// TwinCAT 3 PLC project PLC
// ProgramVersion: 3.1.4024.0
// libraries:
//   EfficientIO Communicator, * (EfficientIO)
//   EfficientIO Energy Basic, * (EfficientIO)
//   EfficientIO ModbusTCP, * (EfficientIO)
//   Lynus Persistent Data V1, * (Lynus AG)
//   Lynus Standards, * (Lynus AG)
//   Tc2_EtherCAT, * (Beckhoff Automation GmbH)
//   Tc2_ModbusSrv, * (Beckhoff Automation GmbH)
//   Tc2_Standard, * (Beckhoff Automation GmbH)
//   Tc2_System, * (Beckhoff Automation GmbH)
//   Tc2_Utilities, * (Beckhoff Automation GmbH)
//   Tc3_Module, * (Beckhoff Automation GmbH)
// project tree:
//   / FastTask.TcTTO, MiddleTask.TcTTO, SlowTask.TcTTO
//   FBs/EL3443_DPM/DUTs/ E_EL3443_DPM_Phase.TcDUT (not stored), E_EL3443_DPM_Total.TcDUT (not stored), MDP5001_341_7CD731EE.TcDUT (not stored), MDP5001_341_I_7CD731EE.TcDUT (not stored), MDP5001_341_O_7CD731EE.TcDUT (not stored), ST_EL3443_DPM_MUX_REAL.TcDUT (not stored), ST_EL3443_DPM_MUX_ULINT.TcDUT (not stored), ST_EL3443_DPM_StatusLx.TcDUT (not stored), ST_EL3443_DPM_StatusTotal.TcDUT (not stored), ST_EL3443_DPM_VariantLx.TcDUT, ST_EL3443_DPM_VariantTotal.TcDUT (not stored), ST_EL3443_DPM_VariantValues.TcDUT (not stored)
//   FBs/EL3443_DPM/ FB_EL3443_DPM.TcPOU (not stored)
//   FBs/EL3446 FW02 or higher/DUTs/ E_EL3446_Phase.TcDUT (not stored), MDP5001_342_066CA8C6.TcDUT, MDP5001_342_I_066CA8C6.TcDUT (not stored), MDP5001_342_O_066CA8C6.TcDUT (not stored), ST_EL3446_MUX_REAL.TcDUT (not stored), ST_EL3446_MUX_ULINT.TcDUT (not stored), ST_EL3446_StatusIx.TcDUT (not stored), ST_EL3446_VariantIx.TcDUT (not stored), ST_EL3446_VariantValues.TcDUT (not stored)
//   FBs/EL3446 FW02 or higher/ FB_EL3446.TcPOU (not stored)
//   FBs/ FB_CoE_EL3443.TcPOU (not stored), FB_CoE_EL3446.TcPOU, FB_ECS_Keba_P30_noWrite.TcPOU, FB_EM_Beckhoff_EL3443.TcPOU, FB_EM_Beckhoff_EL3446.TcPOU, FB_ModBus_100Registers_FC3_inclID.TcPOU, FB_Symo_PV_Inverter_FLOAT_1_DM_30_Inverter_1.TcPOU, FB_Symo_PV_Inverter_INT_1_DM_30_Inverter_1.TcPOU
//   POUs/ prgComEffIO.TcPOU, prgCS.TcPOU, prgEM.TcPOU, prgHW.TcPOU, prgPersistent.TcPOU, prgPV.TcPOU, prgRWEffIO.TcPOU, prgVarEffIO.TcPOU
// real-time tasks:
//   TASK FastTask: cycle T#5ms, priority 19, ADS port 351
//   TASK MiddleTask: cycle T#10ms, priority 20, ADS port 352
//   TASK SlowTask: cycle T#20ms, priority 21, ADS port 353
// I/O:
//   DEVICE Gerät 1 (EtherCAT), AmsNetId 5.114.133.36.2.1
//     Klemme 1 (EK1200) [EK1200-5000 EtherCAT Netzteil (2A E-Bus)]
//       Klemme 2 (EL3443) [EL3443 3K. Leistungsmessung]
//       Klemme 3 (EL3446) [EL3446 DPM 6 K. Strommessklemme]
//       Klemme 4 (EL3446) [EL3446 DPM 6 K. Strommessklemme]
//       Klemme 5 (EL3446) [EL3446 DPM 6 K. Strommessklemme]
//       Klemme 6 (EL3446) [EL3446 DPM 6 K. Strommessklemme]
//       Klemme 7 (EL9011) [EL9011 Endklemme]
// variable links:
//   PLC/PLC Instance <-> Device 1 (EtherCAT)/Term 1 (EK1200)/Term 2 (EL3443)
//     FastTask Inputs/prgHW.MDP5001_341_DPM_Data_Data_{1..20} <-> DPM Data/Data {1..20}  (20 links)
//     FastTask Inputs/prgHW.MDP5001_341_L1_Basic_Current <-> L1 Basic/Current
//     FastTask Inputs/prgHW.MDP5001_341_L2_Basic_Current <-> L2 Basic/Current
//     FastTask Inputs/prgHW.MDP5001_341_L3_Basic_Current <-> L3 Basic/Current
//     FastTask Inputs/prgHW.MDP5001_341_L1_Basic_Voltage <-> L1 Basic/Voltage
//     FastTask Inputs/prgHW.MDP5001_341_L2_Basic_Voltage <-> L2 Basic/Voltage
//     FastTask Inputs/prgHW.MDP5001_341_L3_Basic_Voltage <-> L3 Basic/Voltage
//     FastTask Inputs/prgHW.MDP5001_341_L1_Power_Active_Power <-> L1 Power/Active Power
//     FastTask Inputs/prgHW.MDP5001_341_L2_Power_Active_Power <-> L2 Power/Active Power
//     FastTask Inputs/prgHW.MDP5001_341_L3_Power_Active_Power <-> L3 Power/Active Power
//     FastTask Inputs/prgHW.MDP5001_341_L1_Power_Apparent_Power <-> L1 Power/Apparent Power
//     FastTask Inputs/prgHW.MDP5001_341_L2_Power_Apparent_Power <-> L2 Power/Apparent Power
//     FastTask Inputs/prgHW.MDP5001_341_L3_Power_Apparent_Power <-> L3 Power/Apparent Power
//     FastTask Inputs/prgHW.MDP5001_341_L1_Power_Power_Factor <-> L1 Power/Power Factor
//     FastTask Inputs/prgHW.MDP5001_341_L2_Power_Power_Factor <-> L2 Power/Power Factor
//     FastTask Inputs/prgHW.MDP5001_341_L3_Power_Power_Factor <-> L3 Power/Power Factor
//     FastTask Inputs/prgHW.MDP5001_341_L1_Power_Reactive_Power <-> L1 Power/Reactive Power
//     FastTask Inputs/prgHW.MDP5001_341_L2_Power_Reactive_Power <-> L2 Power/Reactive Power
//     FastTask Inputs/prgHW.MDP5001_341_L3_Power_Reactive_Power <-> L3 Power/Reactive Power
//     FastTask Inputs/prgHW.MDP5001_341_L1_Status_Current_Guard_Error <-> L1 Status/Current Guard Error
//     FastTask Inputs/prgHW.MDP5001_341_L2_Status_Current_Guard_Error <-> L2 Status/Current Guard Error
//     FastTask Inputs/prgHW.MDP5001_341_L3_Status_Current_Guard_Error <-> L3 Status/Current Guard Error
//     FastTask Inputs/prgHW.MDP5001_341_L1_Status_Current_Guard_Warning <-> L1 Status/Current Guard Warning
//     FastTask Inputs/prgHW.MDP5001_341_L2_Status_Current_Guard_Warning <-> L2 Status/Current Guard Warning
//     FastTask Inputs/prgHW.MDP5001_341_L3_Status_Current_Guard_Warning <-> L3 Status/Current Guard Warning
//     FastTask Inputs/prgHW.MDP5001_341_L1_Status_Inaccurate_Current <-> L1 Status/Inaccurate Current
//     FastTask Inputs/prgHW.MDP5001_341_L2_Status_Inaccurate_Current <-> L2 Status/Inaccurate Current
//     FastTask Inputs/prgHW.MDP5001_341_L3_Status_Inaccurate_Current <-> L3 Status/Inaccurate Current
//     FastTask Inputs/prgHW.MDP5001_341_L1_Status_Inaccurate_Voltage <-> L1 Status/Inaccurate Voltage
//     FastTask Inputs/prgHW.MDP5001_341_L2_Status_Inaccurate_Voltage <-> L2 Status/Inaccurate Voltage
//     FastTask Inputs/prgHW.MDP5001_341_L3_Status_Inaccurate_Voltage <-> L3 Status/Inaccurate Voltage
//     FastTask Inputs/prgHW.MDP5001_341_L1_Status_Overcurrent <-> L1 Status/Overcurrent
//     FastTask Inputs/prgHW.MDP5001_341_L2_Status_Overcurrent <-> L2 Status/Overcurrent
//     FastTask Inputs/prgHW.MDP5001_341_L3_Status_Overcurrent <-> L3 Status/Overcurrent
//     FastTask Inputs/prgHW.MDP5001_341_L1_Status_Overvoltage <-> L1 Status/Overvoltage
//     FastTask Inputs/prgHW.MDP5001_341_L2_Status_Overvoltage <-> L2 Status/Overvoltage
//     FastTask Inputs/prgHW.MDP5001_341_L3_Status_Overvoltage <-> L3 Status/Overvoltage
//     FastTask Inputs/prgHW.MDP5001_341_L1_Status_TxPDO_Toggle <-> L1 Status/TxPDO Toggle
//     FastTask Inputs/prgHW.MDP5001_341_L2_Status_TxPDO_Toggle <-> L2 Status/TxPDO Toggle
//     FastTask Inputs/prgHW.MDP5001_341_L3_Status_TxPDO_Toggle <-> L3 Status/TxPDO Toggle
//     FastTask Inputs/prgHW.MDP5001_341_L1_Status_Voltage_Guard_Error <-> L1 Status/Voltage Guard Error
//     FastTask Inputs/prgHW.MDP5001_341_L2_Status_Voltage_Guard_Error <-> L2 Status/Voltage Guard Error
//     FastTask Inputs/prgHW.MDP5001_341_L3_Status_Voltage_Guard_Error <-> L3 Status/Voltage Guard Error
//     FastTask Inputs/prgHW.MDP5001_341_L1_Status_Voltage_Guard_Warning <-> L1 Status/Voltage Guard Warning
//     FastTask Inputs/prgHW.MDP5001_341_L2_Status_Voltage_Guard_Warning <-> L2 Status/Voltage Guard Warning
//     FastTask Inputs/prgHW.MDP5001_341_L3_Status_Voltage_Guard_Warning <-> L3 Status/Voltage Guard Warning
//     FastTask Inputs/prgHW.MDP5001_341_L1_Status_Voltage_Sign_Bit <-> L1 Status/Voltage Sign Bit
//     FastTask Inputs/prgHW.MDP5001_341_L2_Status_Voltage_Sign_Bit <-> L2 Status/Voltage Sign Bit
//     FastTask Inputs/prgHW.MDP5001_341_L3_Status_Voltage_Sign_Bit <-> L3 Status/Voltage Sign Bit
//     FastTask Inputs/prgHW.MDP5001_341_Total_Basic_Calculated_Neutral_Line_Current <-> Total Basic/Calculated Neutral Line Current
//     FastTask Inputs/prgHW.MDP5001_341_Total_Basic_Frequency <-> Total Basic/Frequency
//     FastTask Inputs/prgHW.MDP5001_341_Total_Basic_Power_Factor <-> Total Basic/Power Factor
//     FastTask Inputs/prgHW.MDP5001_341_Total_Status_Active_Power_Guard_Error <-> Total Status/Active Power Guard Error
//     FastTask Inputs/prgHW.MDP5001_341_Total_Status_Active_Power_Guard_Warning <-> Total Status/Active Power Guard Warning
//     FastTask Inputs/prgHW.MDP5001_341_Total_Status_Apparent_Power_Guard_Error <-> Total Status/Apparent Power Guard Error
//     FastTask Inputs/prgHW.MDP5001_341_Total_Status_Apparent_Power_Guard_Warning <-> Total Status/Apparent Power Guard Warning
//     FastTask Inputs/prgHW.MDP5001_341_Total_Status_Frequency_Guard_Error <-> Total Status/Frequency Guard Error
//     FastTask Inputs/prgHW.MDP5001_341_Total_Status_Frequency_Guard_Warning <-> Total Status/Frequency Guard Warning
//     FastTask Inputs/prgHW.MDP5001_341_Total_Status_Grid_Direction <-> Total Status/Grid Direction
//     FastTask Inputs/prgHW.MDP5001_341_Total_Status_Neutral_Current_Guard_Error <-> Total Status/Neutral Current Guard Error
//     FastTask Inputs/prgHW.MDP5001_341_Total_Status_Neutral_Current_Guard_Warning <-> Total Status/Neutral Current Guard Warning
//     FastTask Inputs/prgHW.MDP5001_341_Total_Status_Power_Quality_Factor <-> Total Status/Power Quality Factor
//     FastTask Inputs/prgHW.MDP5001_341_Total_Status_Power_Quality_Guard_Error <-> Total Status/Power Quality Guard Error
//     FastTask Inputs/prgHW.MDP5001_341_Total_Status_Power_Quality_Guard_Warning <-> Total Status/Power Quality Guard Warning
//     FastTask Inputs/prgHW.MDP5001_341_Total_Status_System_State <-> Total Status/System State
//     FastTask Inputs/prgHW.MDP5001_341_Total_Status_TxPDO_State <-> Total Status/TxPDO State
//     FastTask Inputs/prgHW.MDP5001_341_Total_Status_TxPDO_Toggle <-> Total Status/TxPDO Toggle
//     FastTask Inputs/prgHW.MDP5001_341_Total_Variant_Value_In_Index_1_REAL <-> Total Variant Value In/Index 1 REAL
//     FastTask Inputs/prgHW.MDP5001_341_Total_Variant_Value_In_Index_2_REAL <-> Total Variant Value In/Index 2 REAL
//     FastTask Inputs/prgHW.MDP5001_341_Total_Variant_Value_In_Index_3_REAL <-> Total Variant Value In/Index 3 REAL
//     FastTask Inputs/prgHW.MDP5001_341_Total_Variant_Value_In_Index_4_ULINT <-> Total Variant Value In/Index 4 ULINT
//     FastTask Inputs/prgHW.MDP5001_341_Total_Variant_Value_In_TxPDO_Toggle <-> Total Variant Value In/TxPDO Toggle
//     FastTask Inputs/prgHW.MDP5001_341_Total_Variant_Value_In_Value_1_REAL <-> Total Variant Value In/Value 1 REAL
//     FastTask Inputs/prgHW.MDP5001_341_Total_Variant_Value_In_Value_2_REAL <-> Total Variant Value In/Value 2 REAL
//     FastTask Inputs/prgHW.MDP5001_341_Total_Variant_Value_In_Value_3_REAL <-> Total Variant Value In/Value 3 REAL
//     FastTask Inputs/prgHW.MDP5001_341_Total_Variant_Value_In_Value_4_ULINT <-> Total Variant Value In/Value 4 ULINT
//     FastTask Outputs/prgHW.MDP5001_341_Total_Interval_Reset_Interval <-> Total Interval/Reset Interval
//     FastTask Outputs/prgHW.MDP5001_341_Total_Variant_Value_Out_Index_1_REAL <-> Total Variant Value Out/Index 1 REAL
//     FastTask Outputs/prgHW.MDP5001_341_Total_Variant_Value_Out_Index_2_REAL <-> Total Variant Value Out/Index 2 REAL
//     FastTask Outputs/prgHW.MDP5001_341_Total_Variant_Value_Out_Index_3_REAL <-> Total Variant Value Out/Index 3 REAL
//     FastTask Outputs/prgHW.MDP5001_341_Total_Variant_Value_Out_Index_4_ULINT <-> Total Variant Value Out/Index 4 ULINT
//   PLC/PLC Instance <-> Device 1 (EtherCAT)/Term 1 (EK1200)/Term 3 (EL3446)
//     FastTask Inputs/prgHW.MDP5001_342_DPM_Variant_Value_In_Index_1_REAL_1 <-> DPM Variant Value In/Index 1 REAL
//     FastTask Inputs/prgHW.MDP5001_342_DPM_Variant_Value_In_Index_2_REAL_1 <-> DPM Variant Value In/Index 2 REAL
//     FastTask Inputs/prgHW.MDP5001_342_DPM_Variant_Value_In_Index_3_REAL_1 <-> DPM Variant Value In/Index 3 REAL
//     FastTask Inputs/prgHW.MDP5001_342_DPM_Variant_Value_In_Index_4_ULINT_1 <-> DPM Variant Value In/Index 4 ULINT
//     FastTask Inputs/prgHW.MDP5001_342_DPM_Variant_Value_In_TxPDO_Toggle_1 <-> DPM Variant Value In/TxPDO Toggle
//     FastTask Inputs/prgHW.MDP5001_342_DPM_Variant_Value_In_Value_1_REAL_1 <-> DPM Variant Value In/Value 1 REAL
//     FastTask Inputs/prgHW.MDP5001_342_DPM_Variant_Value_In_Value_2_REAL_1 <-> DPM Variant Value In/Value 2 REAL
//     FastTask Inputs/prgHW.MDP5001_342_DPM_Variant_Value_In_Value_3_REAL_1 <-> DPM Variant Value In/Value 3 REAL
//     FastTask Inputs/prgHW.MDP5001_342_DPM_Variant_Value_In_Value_4_ULINT_1 <-> DPM Variant Value In/Value 4 ULINT
//     FastTask Inputs/prgHW.MDP5001_342_I{1..6}_Channel_Active_Energy_1 <-> I{1..6} Channel/Active Energy  (6 links)
//     FastTask Inputs/prgHW.MDP5001_342_I{1..6}_Channel_Active_Power_1 <-> I{1..6} Channel/Active Power  (6 links)
//     FastTask Inputs/prgHW.MDP5001_342_I{1..6}_Channel_Active_Power_Guard_Error_1 <-> I{1..6} Channel/Active Power Guard Error  (6 links)
//     FastTask Inputs/prgHW.MDP5001_342_I{1..6}_Channel_Active_Power_Guard_Warning_1 <-> I{1..6} Channel/Active Power Guard Warning  (6 links)
//     FastTask Inputs/prgHW.MDP5001_342_I{1..6}_Channel_Apparent_Power_1 <-> I{1..6} Channel/Apparent Power  (6 links)
//     FastTask Inputs/prgHW.MDP5001_342_I{1..6}_Channel_Apparent_Power_Guard_Error_1 <-> I{1..6} Channel/Apparent Power Guard Error  (6 links)
//     FastTask Inputs/prgHW.MDP5001_342_I{1..6}_Channel_Apparent_Power_Guard_Warning_1 <-> I{1..6} Channel/Apparent Power Guard Warning  (6 links)
//     FastTask Inputs/prgHW.MDP5001_342_I{1..6}_Channel_Current_1 <-> I{1..6} Channel/Current  (6 links)
//     FastTask Inputs/prgHW.MDP5001_342_I{1..6}_Channel_Current_Guard_Error_1 <-> I{1..6} Channel/Current Guard Error  (6 links)
//     FastTask Inputs/prgHW.MDP5001_342_I{1..6}_Channel_Current_Guard_Warning_1 <-> I{1..6} Channel/Current Guard Warning  (6 links)
//     FastTask Inputs/prgHW.MDP5001_342_I{1..6}_Channel_DPM_Inaccurate_1 <-> I{1..6} Channel/DPM Inaccurate  (6 links)
//     FastTask Inputs/prgHW.MDP5001_342_I{1..6}_Channel_DPM_Timeout_1 <-> I{1..6} Channel/DPM Timeout  (6 links)
//     FastTask Inputs/prgHW.MDP5001_342_I{1..6}_Channel_Inaccurate_Current_1 <-> I{1..6} Channel/Inaccurate Current  (6 links)
//     FastTask Inputs/prgHW.MDP5001_342_I{1..6}_Channel_Overcurrent_1 <-> I{1..6} Channel/Overcurrent  (6 links)
//     FastTask Inputs/prgHW.MDP5001_342_I{1..6}_Channel_Reactive_Power_Fundamental_1 <-> I{1..6} Channel/Reactive Power Fundamental  (6 links)
//     FastTask Inputs/prgHW.MDP5001_342_I{1..6}_Channel_Reactive_Power_Guard_Error_1 <-> I{1..6} Channel/Reactive Power Guard Error  (6 links)
//     FastTask Inputs/prgHW.MDP5001_342_I{1..6}_Channel_Reactive_Power_Guard_Warning_1 <-> I{1..6} Channel/Reactive Power Guard Warning  (6 links)
//     FastTask Inputs/prgHW.MDP5001_342_I{1..6}_Channel_TxPDO_Toggle_1 <-> I{1..6} Channel/TxPDO Toggle  (6 links)
//     FastTask Outputs/prgHW.MDP5001_342_DPM_Data_Data_{1..20}_1 <-> DPM Data/Data {1..20}  (20 links)
//     FastTask Outputs/prgHW.MDP5001_342_DPM_Variant_Value_Out_Index_1_REAL_1 <-> DPM Variant Value Out/Index 1 REAL
//     FastTask Outputs/prgHW.MDP5001_342_DPM_Variant_Value_Out_Index_2_REAL_1 <-> DPM Variant Value Out/Index 2 REAL
//     FastTask Outputs/prgHW.MDP5001_342_DPM_Variant_Value_Out_Index_3_REAL_1 <-> DPM Variant Value Out/Index 3 REAL
//     FastTask Outputs/prgHW.MDP5001_342_DPM_Variant_Value_Out_Index_4_ULINT_1 <-> DPM Variant Value Out/Index 4 ULINT
//   PLC/PLC Instance <-> Device 1 (EtherCAT)/Term 1 (EK1200)/Term 4 (EL3446)
//     FastTask Inputs/prgHW.MDP5001_342_DPM_Variant_Value_In_Index_1_REAL_2 <-> DPM Variant Value In/Index 1 REAL
//     FastTask Inputs/prgHW.MDP5001_342_DPM_Variant_Value_In_Index_2_REAL_2 <-> DPM Variant Value In/Index 2 REAL
//     FastTask Inputs/prgHW.MDP5001_342_DPM_Variant_Value_In_Index_3_REAL_2 <-> DPM Variant Value In/Index 3 REAL
//     FastTask Inputs/prgHW.MDP5001_342_DPM_Variant_Value_In_Index_4_ULINT_2 <-> DPM Variant Value In/Index 4 ULINT
//     FastTask Inputs/prgHW.MDP5001_342_DPM_Variant_Value_In_TxPDO_Toggle_2 <-> DPM Variant Value In/TxPDO Toggle
//     FastTask Inputs/prgHW.MDP5001_342_DPM_Variant_Value_In_Value_1_REAL_2 <-> DPM Variant Value In/Value 1 REAL
//     FastTask Inputs/prgHW.MDP5001_342_DPM_Variant_Value_In_Value_2_REAL_2 <-> DPM Variant Value In/Value 2 REAL
//     FastTask Inputs/prgHW.MDP5001_342_DPM_Variant_Value_In_Value_3_REAL_2 <-> DPM Variant Value In/Value 3 REAL
//     FastTask Inputs/prgHW.MDP5001_342_DPM_Variant_Value_In_Value_4_ULINT_2 <-> DPM Variant Value In/Value 4 ULINT
//     FastTask Inputs/prgHW.MDP5001_342_I{1..6}_Channel_Active_Energy_2 <-> I{1..6} Channel/Active Energy  (6 links)
//     FastTask Inputs/prgHW.MDP5001_342_I{1..6}_Channel_Active_Power_2 <-> I{1..6} Channel/Active Power  (6 links)
//     FastTask Inputs/prgHW.MDP5001_342_I{1..6}_Channel_Active_Power_Guard_Error_2 <-> I{1..6} Channel/Active Power Guard Error  (6 links)
//     FastTask Inputs/prgHW.MDP5001_342_I{1..6}_Channel_Active_Power_Guard_Warning_2 <-> I{1..6} Channel/Active Power Guard Warning  (6 links)
//     FastTask Inputs/prgHW.MDP5001_342_I{1..6}_Channel_Apparent_Power_2 <-> I{1..6} Channel/Apparent Power  (6 links)
//     FastTask Inputs/prgHW.MDP5001_342_I{1..6}_Channel_Apparent_Power_Guard_Error_2 <-> I{1..6} Channel/Apparent Power Guard Error  (6 links)
//     FastTask Inputs/prgHW.MDP5001_342_I{1..6}_Channel_Apparent_Power_Guard_Warning_2 <-> I{1..6} Channel/Apparent Power Guard Warning  (6 links)
//     FastTask Inputs/prgHW.MDP5001_342_I{1..6}_Channel_Current_2 <-> I{1..6} Channel/Current  (6 links)
//     FastTask Inputs/prgHW.MDP5001_342_I{1..6}_Channel_Current_Guard_Error_2 <-> I{1..6} Channel/Current Guard Error  (6 links)
//     FastTask Inputs/prgHW.MDP5001_342_I{1..6}_Channel_Current_Guard_Warning_2 <-> I{1..6} Channel/Current Guard Warning  (6 links)
//     FastTask Inputs/prgHW.MDP5001_342_I{1..6}_Channel_DPM_Inaccurate_2 <-> I{1..6} Channel/DPM Inaccurate  (6 links)
//     FastTask Inputs/prgHW.MDP5001_342_I{1..6}_Channel_DPM_Timeout_2 <-> I{1..6} Channel/DPM Timeout  (6 links)
//     FastTask Inputs/prgHW.MDP5001_342_I{1..6}_Channel_Inaccurate_Current_2 <-> I{1..6} Channel/Inaccurate Current  (6 links)
//     FastTask Inputs/prgHW.MDP5001_342_I{1..6}_Channel_Overcurrent_2 <-> I{1..6} Channel/Overcurrent  (6 links)
//     FastTask Inputs/prgHW.MDP5001_342_I{1..6}_Channel_Reactive_Power_Fundamental_2 <-> I{1..6} Channel/Reactive Power Fundamental  (6 links)
//     FastTask Inputs/prgHW.MDP5001_342_I{1..6}_Channel_Reactive_Power_Guard_Error_2 <-> I{1..6} Channel/Reactive Power Guard Error  (6 links)
//     FastTask Inputs/prgHW.MDP5001_342_I{1..6}_Channel_Reactive_Power_Guard_Warning_2 <-> I{1..6} Channel/Reactive Power Guard Warning  (6 links)
//     FastTask Inputs/prgHW.MDP5001_342_I{1..6}_Channel_TxPDO_Toggle_2 <-> I{1..6} Channel/TxPDO Toggle  (6 links)
//     FastTask Outputs/prgHW.MDP5001_342_DPM_Data_Data_{1..20}_2 <-> DPM Data/Data {1..20}  (20 links)
//     FastTask Outputs/prgHW.MDP5001_342_DPM_Variant_Value_Out_Index_1_REAL_2 <-> DPM Variant Value Out/Index 1 REAL
//     FastTask Outputs/prgHW.MDP5001_342_DPM_Variant_Value_Out_Index_2_REAL_2 <-> DPM Variant Value Out/Index 2 REAL
//     FastTask Outputs/prgHW.MDP5001_342_DPM_Variant_Value_Out_Index_3_REAL_2 <-> DPM Variant Value Out/Index 3 REAL
//     FastTask Outputs/prgHW.MDP5001_342_DPM_Variant_Value_Out_Index_4_ULINT_2 <-> DPM Variant Value Out/Index 4 ULINT
//   PLC/PLC Instance <-> Device 1 (EtherCAT)/Term 1 (EK1200)/Term 5 (EL3446)
//     FastTask Inputs/prgHW.MDP5001_342_DPM_Variant_Value_In_Index_1_REAL_3 <-> DPM Variant Value In/Index 1 REAL
//     FastTask Inputs/prgHW.MDP5001_342_DPM_Variant_Value_In_Index_2_REAL_3 <-> DPM Variant Value In/Index 2 REAL
//     FastTask Inputs/prgHW.MDP5001_342_DPM_Variant_Value_In_Index_3_REAL_3 <-> DPM Variant Value In/Index 3 REAL
//     FastTask Inputs/prgHW.MDP5001_342_DPM_Variant_Value_In_Index_4_ULINT_3 <-> DPM Variant Value In/Index 4 ULINT
//     FastTask Inputs/prgHW.MDP5001_342_DPM_Variant_Value_In_TxPDO_Toggle_3 <-> DPM Variant Value In/TxPDO Toggle
//     FastTask Inputs/prgHW.MDP5001_342_DPM_Variant_Value_In_Value_1_REAL_3 <-> DPM Variant Value In/Value 1 REAL
//     FastTask Inputs/prgHW.MDP5001_342_DPM_Variant_Value_In_Value_2_REAL_3 <-> DPM Variant Value In/Value 2 REAL
//     FastTask Inputs/prgHW.MDP5001_342_DPM_Variant_Value_In_Value_3_REAL_3 <-> DPM Variant Value In/Value 3 REAL
//     FastTask Inputs/prgHW.MDP5001_342_DPM_Variant_Value_In_Value_4_ULINT_3 <-> DPM Variant Value In/Value 4 ULINT
//     FastTask Inputs/prgHW.MDP5001_342_I{1..6}_Channel_Active_Energy_3 <-> I{1..6} Channel/Active Energy  (6 links)
//     FastTask Inputs/prgHW.MDP5001_342_I{1..6}_Channel_Active_Power_3 <-> I{1..6} Channel/Active Power  (6 links)
//     FastTask Inputs/prgHW.MDP5001_342_I{1..6}_Channel_Active_Power_Guard_Error_3 <-> I{1..6} Channel/Active Power Guard Error  (6 links)
//     FastTask Inputs/prgHW.MDP5001_342_I{1..6}_Channel_Active_Power_Guard_Warning_3 <-> I{1..6} Channel/Active Power Guard Warning  (6 links)
//     FastTask Inputs/prgHW.MDP5001_342_I{1..6}_Channel_Apparent_Power_3 <-> I{1..6} Channel/Apparent Power  (6 links)
//     FastTask Inputs/prgHW.MDP5001_342_I{1..6}_Channel_Apparent_Power_Guard_Error_3 <-> I{1..6} Channel/Apparent Power Guard Error  (6 links)
//     FastTask Inputs/prgHW.MDP5001_342_I{1..6}_Channel_Apparent_Power_Guard_Warning_3 <-> I{1..6} Channel/Apparent Power Guard Warning  (6 links)
//     FastTask Inputs/prgHW.MDP5001_342_I{1..6}_Channel_Current_3 <-> I{1..6} Channel/Current  (6 links)
//     FastTask Inputs/prgHW.MDP5001_342_I{1..6}_Channel_Current_Guard_Error_3 <-> I{1..6} Channel/Current Guard Error  (6 links)
//     FastTask Inputs/prgHW.MDP5001_342_I{1..6}_Channel_Current_Guard_Warning_3 <-> I{1..6} Channel/Current Guard Warning  (6 links)
//     FastTask Inputs/prgHW.MDP5001_342_I{1..6}_Channel_DPM_Inaccurate_3 <-> I{1..6} Channel/DPM Inaccurate  (6 links)
//     FastTask Inputs/prgHW.MDP5001_342_I{1..6}_Channel_DPM_Timeout_3 <-> I{1..6} Channel/DPM Timeout  (6 links)
//     FastTask Inputs/prgHW.MDP5001_342_I{1..6}_Channel_Inaccurate_Current_3 <-> I{1..6} Channel/Inaccurate Current  (6 links)
//     FastTask Inputs/prgHW.MDP5001_342_I{1..6}_Channel_Overcurrent_3 <-> I{1..6} Channel/Overcurrent  (6 links)
//     FastTask Inputs/prgHW.MDP5001_342_I{1..6}_Channel_Reactive_Power_Fundamental_3 <-> I{1..6} Channel/Reactive Power Fundamental  (6 links)
//     FastTask Inputs/prgHW.MDP5001_342_I{1..6}_Channel_Reactive_Power_Guard_Error_3 <-> I{1..6} Channel/Reactive Power Guard Error  (6 links)
//     FastTask Inputs/prgHW.MDP5001_342_I{1..6}_Channel_Reactive_Power_Guard_Warning_3 <-> I{1..6} Channel/Reactive Power Guard Warning  (6 links)
//     FastTask Inputs/prgHW.MDP5001_342_I{1..6}_Channel_TxPDO_Toggle_3 <-> I{1..6} Channel/TxPDO Toggle  (6 links)
//     FastTask Outputs/prgHW.MDP5001_342_DPM_Data_Data_{1..20}_3 <-> DPM Data/Data {1..20}  (20 links)
//     FastTask Outputs/prgHW.MDP5001_342_DPM_Variant_Value_Out_Index_1_REAL_3 <-> DPM Variant Value Out/Index 1 REAL
//     FastTask Outputs/prgHW.MDP5001_342_DPM_Variant_Value_Out_Index_2_REAL_3 <-> DPM Variant Value Out/Index 2 REAL
//     FastTask Outputs/prgHW.MDP5001_342_DPM_Variant_Value_Out_Index_3_REAL_3 <-> DPM Variant Value Out/Index 3 REAL
//     FastTask Outputs/prgHW.MDP5001_342_DPM_Variant_Value_Out_Index_4_ULINT_3 <-> DPM Variant Value Out/Index 4 ULINT
//   PLC/PLC Instance <-> Device 1 (EtherCAT)/Term 1 (EK1200)/Term 6 (EL3446)
//     FastTask Inputs/prgHW.MDP5001_442_DPM_Variant_Value_In_Index_1_REAL_4 <-> DPM Variant Value In/Index 1 REAL
//     FastTask Inputs/prgHW.MDP5001_442_DPM_Variant_Value_In_Index_2_REAL_4 <-> DPM Variant Value In/Index 2 REAL
//     FastTask Inputs/prgHW.MDP5001_442_DPM_Variant_Value_In_Index_3_REAL_4 <-> DPM Variant Value In/Index 3 REAL
//     FastTask Inputs/prgHW.MDP5001_442_DPM_Variant_Value_In_Index_4_ULINT_4 <-> DPM Variant Value In/Index 4 ULINT
//     FastTask Inputs/prgHW.MDP5001_442_DPM_Variant_Value_In_TxPDO_Toggle_4 <-> DPM Variant Value In/TxPDO Toggle
//     FastTask Inputs/prgHW.MDP5001_442_DPM_Variant_Value_In_Value_1_REAL_4 <-> DPM Variant Value In/Value 1 REAL
//     FastTask Inputs/prgHW.MDP5001_442_DPM_Variant_Value_In_Value_2_REAL_4 <-> DPM Variant Value In/Value 2 REAL
//     FastTask Inputs/prgHW.MDP5001_442_DPM_Variant_Value_In_Value_3_REAL_4 <-> DPM Variant Value In/Value 3 REAL
//     FastTask Inputs/prgHW.MDP5001_442_DPM_Variant_Value_In_Value_4_ULINT_4 <-> DPM Variant Value In/Value 4 ULINT
//     FastTask Inputs/prgHW.MDP5001_442_I{1..6}_Channel_Active_Energy_4 <-> I{1..6} Channel/Active Energy  (6 links)
//     FastTask Inputs/prgHW.MDP5001_442_I{1..6}_Channel_Active_Power_4 <-> I{1..6} Channel/Active Power  (6 links)
//     FastTask Inputs/prgHW.MDP5001_442_I{1..6}_Channel_Active_Power_Guard_Error_4 <-> I{1..6} Channel/Active Power Guard Error  (6 links)
//     FastTask Inputs/prgHW.MDP5001_442_I{1..6}_Channel_Active_Power_Guard_Warning_4 <-> I{1..6} Channel/Active Power Guard Warning  (6 links)
//     FastTask Inputs/prgHW.MDP5001_442_I{1..6}_Channel_Apparent_Power_4 <-> I{1..6} Channel/Apparent Power  (6 links)
//     FastTask Inputs/prgHW.MDP5001_442_I{1..6}_Channel_Apparent_Power_Guard_Error_4 <-> I{1..6} Channel/Apparent Power Guard Error  (6 links)
//     FastTask Inputs/prgHW.MDP5001_442_I{1..6}_Channel_Apparent_Power_Guard_Warning_4 <-> I{1..6} Channel/Apparent Power Guard Warning  (6 links)
//     FastTask Inputs/prgHW.MDP5001_442_I{1..6}_Channel_Current_4 <-> I{1..6} Channel/Current  (6 links)
//     FastTask Inputs/prgHW.MDP5001_442_I{1..6}_Channel_Current_Guard_Error_4 <-> I{1..6} Channel/Current Guard Error  (6 links)
//     FastTask Inputs/prgHW.MDP5001_442_I{1..6}_Channel_Current_Guard_Warning_4 <-> I{1..6} Channel/Current Guard Warning  (6 links)
//     FastTask Inputs/prgHW.MDP5001_442_I{1..6}_Channel_DPM_Inaccurate_4 <-> I{1..6} Channel/DPM Inaccurate  (6 links)
//     FastTask Inputs/prgHW.MDP5001_442_I{1..6}_Channel_DPM_Timeout_4 <-> I{1..6} Channel/DPM Timeout  (6 links)
//     FastTask Inputs/prgHW.MDP5001_442_I{1..6}_Channel_Inaccurate_Current_4 <-> I{1..6} Channel/Inaccurate Current  (6 links)
//     FastTask Inputs/prgHW.MDP5001_442_I{1..6}_Channel_Overcurrent_4 <-> I{1..6} Channel/Overcurrent  (6 links)
//     FastTask Inputs/prgHW.MDP5001_442_I{1..6}_Channel_Reactive_Power_Fundamental_4 <-> I{1..6} Channel/Reactive Power Fundamental  (6 links)
//     FastTask Inputs/prgHW.MDP5001_442_I{1..6}_Channel_Reactive_Power_Guard_Error_4 <-> I{1..6} Channel/Reactive Power Guard Error  (6 links)
//     FastTask Inputs/prgHW.MDP5001_442_I{1..6}_Channel_Reactive_Power_Guard_Warning_4 <-> I{1..6} Channel/Reactive Power Guard Warning  (6 links)
//     FastTask Inputs/prgHW.MDP5001_442_I{1..6}_Channel_TxPDO_Toggle_4 <-> I{1..6} Channel/TxPDO Toggle  (6 links)
//     FastTask Outputs/prgHW.MDP5001_342_DPM_Data_Data_{1..20}_4 <-> DPM Data/Data {1..20}  (20 links)
//     FastTask Outputs/prgHW.MDP5001_342_DPM_Variant_Value_Out_Index_1_REAL_4 <-> DPM Variant Value Out/Index 1 REAL
//     FastTask Outputs/prgHW.MDP5001_342_DPM_Variant_Value_Out_Index_2_REAL_4 <-> DPM Variant Value Out/Index 2 REAL
//     FastTask Outputs/prgHW.MDP5001_342_DPM_Variant_Value_Out_Index_3_REAL_4 <-> DPM Variant Value Out/Index 3 REAL
//     FastTask Outputs/prgHW.MDP5001_342_DPM_Variant_Value_Out_Index_4_ULINT_4 <-> DPM Variant Value Out/Index 4 ULINT

CONFIGURATION PLC
    RESOURCE PLC ON TwinCAT3
        TASK FastTask(INTERVAL := T#5ms, PRIORITY := 19);
        TASK MiddleTask(INTERVAL := T#10ms, PRIORITY := 20);
        TASK SlowTask(INTERVAL := T#20ms, PRIORITY := 21);
        PROGRAM prgVarEffIO WITH FastTask : prgVarEffIO;
        PROGRAM prgRWEffIO WITH FastTask : prgRWEffIO;
        PROGRAM prgPersistent WITH FastTask : prgPersistent;
        PROGRAM prgHW WITH FastTask : prgHW;
        PROGRAM prgEM WITH MiddleTask : prgEM;
        PROGRAM prgPV WITH MiddleTask : prgPV;
        PROGRAM prgCS WITH MiddleTask : prgCS;
        PROGRAM prgComEffIO WITH SlowTask : prgComEffIO;
    END_RESOURCE
END_CONFIGURATION

// ---- FBs/EL3443_DPM/DUTs/ST_EL3443_DPM_VariantLx.TcDUT
TYPE ST_EL3443_DPM_VariantLx :
STRUCT
    fU_RMS : REAL;						// [V] (Real Selector: 1 (Examp.: 257 = 1 + 256 for ch. 1)) RMS value of the voltage
    fU_peak : REAL;						// [V] (Real Selector: 2 (Examp.: 770 = 2 + 768 for ch. 3)) Peak value of the instantaneous voltage in the last interval
    nU_Last_Zero_Cross : ULINT;			// [V] (UINT Selector: 3) DC time of the penultimate voltage zero crossing
    fU_RMS_Minimum : REAL;				// [V] (Real Selector: 4) Minimum RMS value of the voltage in the last interval
    fU_RMS_Maximum : REAL;				// [V] (Real Selector: 5) Maximum RMS value of the voltage in the last interval
    fULL : REAL;						// [V] (Real Selector: 6) RMS value of the phase-to-phase voltage (Channel 1: U_L1L2; Channel 1: U_L2L3; Channel 3: U_L3L1) 
    fI_RMS : REAL;						// [A] (Real Selector: 8) RMS value of the current
    fI_peak : REAL;						// [A] (Real Selector: 9) Peak value of the instantaneous current in the last interval
    fI_RMS_Minimum : REAL;				// [A] (Real Selector: 11) Minimum RMS value of the current in the last interval
    fI_RMS_Maximum : REAL;				// [A] (Real Selector: 12) Maximum RMS value of the current in the last interval
    fFrequency : REAL;					// [Hz] (Real Selector: 17) Frequency of this phase
    fPhi : REAL;						// [°] (Real Selector: 21) Phase angle of the fundamental wave
    fCOS_phi : REAL;					// [-] (Real Selector: 22) Cosine of the fundamental wave phase angle
    fPower_Factor : REAL;				// [-] (Real Selector: 23) Power factor
    fP : REAL;							// [W] (Real Selector: 26) Active power
    fPavg : REAL;						// [W] (Real Selector: 27) Average active power during the last interval
    fPmin : REAL;						// [W] (Real Selector: 28) Minimum active power in the last interval
    fPmax : REAL;						// [W] (Real Selector: 29) Maximum active power in the last interval
    fS : REAL;							// [VA] (Real Selector: 32) Apparent power
    fSavg : REAL;						// [VA] (Real Selector: 33) Average apparent power during the last interval
    fSmin : REAL;						// [VA] (Real Selector: 34) Minimum apparent power in last interval
    fSmax : REAL;						// [VA] (Real Selector: 35) Minimum apparent power in last interval
    fQ : REAL;							// [Var] (Real Selector: 38) Reactive power
    fQavg : REAL;						// [Var] (Real Selector: 39) Average reactive power average during the last interval
    fQmin : REAL;						// [Var] (Real Selector: 40) Minimum reactive power in the last interval
    fQmax : REAL;						// [Var] (Real Selector: 41) Maximum reactive power in the last interval
    nEP : LINT;							// [mhW] (LINT Selector: 45) Recorded active energy
    nEP_pos : ULINT;					// [mhW] (UINT Selector: 46) Received active energy
    nEP_neg : ULINT;					// [mhW] (UINT Selector: 47) Supplied active energy
	nEP_interval : LINT;				// [mhW] (LINT Selector: 48) Recorded active energy in the last interval
	nEP_pos_interval : ULINT;			// [mhW] (UINT Selector: 49) Received active energy in the last interval
	nEP_neg_interval : ULINT;			// [mhW] (UINT Selector: 50) Supplied active energy in the last interval
    nES : LINT;							// [mhW] (LINT Selector: 51) Apparent energy
    nES_pos : ULINT;					// [mhW] (UINT Selector: 52) Apparent energy
    nES_neg : ULINT;					// [mhW] (UINT Selector: 53) Apparent energy
	nES_interval : LINT;				// [mhW] (LINT Selector: 54) Apparent energy in the last interval
	nES_pos_interval : ULINT;			// [mhW] (UINT Selector: 55) Apparent energy in the last interval
	nES_neg_interval : ULINT;			// [mhW] (UINT Selector: 56) Apparent energy in the last interval
    nEQ : LINT;							// [mhW] (LINT Selector: 57) Reactive energy
    nEQ_pos : ULINT;					// [mhW] (UINT Selector: 58) Reactive energy
    nEQ_neg : ULINT;					// [mhW] (UINT Selector: 59) Reactive energy
	nEQ_interval : LINT;				// [mhW] (LINT Selector: 60) Reactive energy in the last interval
	nEQ_pos_interval : ULINT;			// [mhW] (UINT Selector: 62) Reactive energy in the last interval
	nEQ_neg_interval : ULINT;			// [mhW] (UINT Selector: 63) Reactive energy in the last interval
    fTHD_U : REAL;						// [-] (Real Selector: 95) "Total Harmonic Distortion" is the distortion factor of the voltage. It indicates the ratio of the harmonic components of an oscillation relative to its fundamental.
    fRMS_fund_U : REAL;					// [V] (Real Selector: 98) Amplitude of the fundamental wave
    fF_Ref_U : REAL;					// [Hz] (Real Selector: 99) Reference frequency of the voltage harmonic: Specifies the underlying fundamental frequency, e.g.: 50 or 60 Hz.
    fHarmonics_U : ARRAY [0..41] OF REAL;// [% of the fundamental wave] (Real Selector: 100-141) 0 => DC component, 1 => fundamental wave, 2=> 2nd harmonic, 3=> 3rd harmonic
    fTHD_I : REAL;						// [-] (Real Selector: 165) "Total Harmonic Distortion" is the distortion factor of the current. It indicates the ratio of the harmonic components of an oscillation relative to its fundamental.
    fTDD_I : REAL;						// [% of the maximum current] (Real Selector: 166) "Total Demand Distortion" indicates the ratio between the current harmonics and the maximum current (EL3443: 1A and EL3443-0010: 5A)
    fRMS_fund_I : REAL;					// [A] (Real Selector: 168) Amplitude of the fundamental wave
    fF_Ref_I : REAL;					// [Hz] (Real Selector: 169) Reference frequency of the current harmonic: Specifies the underlying fundamental frequency, e.g.: 50 or 60 Hz.
    fHarmonics_I : ARRAY [0..41] OF REAL;// [% of the fundamental wave] (Real Selector: 170-211) 0 => DC component, 1 => fundamental wave, 2=> 2nd harmonic, 3=> 3rd harmonic
END_STRUCT
END_TYPE

// ---- FBs/EL3446 FW02 or higher/DUTs/MDP5001_342_066CA8C6.TcDUT
TYPE MDP5001_342_066CA8C6 :
STRUCT
	MDP5001_342_Input	: MDP5001_342_I_066CA8C6;
	MDP5001_342_Output	: MDP5001_342_O_066CA8C6;
END_STRUCT
END_TYPE

// ---- POUs/prgVarEffIO.TcPOU
PROGRAM prgVarEffIO
VAR
	fbVar		: FB_VarInfo;
END_VAR

fbVar(
	bReadInfo:= , 
	eTMCFile:= eSelectTMCFile.eUseTMCFile, 
	eSavePositionTMCFile:= eSavePositionOnPLC.ePostionC, 
	udiCounterFoundVariables=> , 
	bError=> , 
	bBusy=> , 
	byProgress=> , 
	udiErrorCodeOut=> , 
	eErrorVarInfo_Out=> , 
	sVarWithError=> );
fbVar();
fbVar();

END_PROGRAM

// ---- POUs/prgRWEffIO.TcPOU
PROGRAM prgRWEffIO
VAR
	fbRW1		: FB_ReadWrite_V2;
	fbRW2		: FB_ReadWrite_V2;
	fbRW3		: FB_ReadWrite_V2;
END_VAR

fbRW1(	eUploadType := eSelectDataUploadType.e_Change_Intervall5min,
		bBusy=> , 
		bError=> , 
		udiErrorCodeOut=> , 
		eErrorReadWrite_Out=> );
fbRW2(	eUploadType := eSelectDataUploadType.e_Change_noIntervall,
		bBusy=> , 
		bError=> , 
		udiErrorCodeOut=> , 
		eErrorReadWrite_Out=> );		
fbRW3(	eUploadType := eSelectDataUploadType.e_Change_noIntervall,
		bBusy=> , 
		bError=> , 
		udiErrorCodeOut=> , 
		eErrorReadWrite_Out=> );

END_PROGRAM

// ---- POUs/prgPersistent.TcPOU
PROGRAM prgPersistent
VAR
	fbUSV		: FB_WritePersistentData_CX81xx;
	
	fb_Reboot		: NT_reboot;
	m_Reboot		: BOOL:=FALSE;
	Int_LiveCount_1min	:INT; 							//{#lynus.ag#()}
	ton_LiveCount	:TON;	
	int_liveCount		:INT;				//{#lynus.ag#()}
END_VAR

(*
fbUSV(
	eSaveModeData:= eUSVSaveMode.eSaveWhenPowerfail, 
	bLoadPersistentDataOk=> , 
	bPowerFailDetect=> , 
	bError=> , 
	bySaveProcess=> , 
	dwStorageLast24h=> , 
	udiErrorCode=> );
*)	
	
fb_Reboot(	netid := '',
			delay := 2,
			start := m_Reboot);

// 1 min live count
ton_LiveCount(PT:=T#1M);
IF ton_LiveCount.Q THEN
	Int_LiveCount_1min := Int_LiveCount_1min + 1;
	ton_LiveCount.IN := FALSE;
ELSE
	ton_LiveCount.IN := TRUE;
END_IF
// livecount
int_liveCount := int_liveCount+1;

END_PROGRAM

// ---- POUs/prgHW.TcPOU
PROGRAM prgHW
VAR
	// IOs for EL3443
	{attribute 'TcLinkTo' := 'TIID^Gerät 1 (EtherCAT)^Klemme 1 (EK1200)^Klemme 2 (EL3443)^L1 Status^Voltage Sign Bit'}
	MDP5001_341_L1_Status_Voltage_Sign_Bit   	AT%I*  : BOOL;  // linked via attribute 
	{attribute 'TcLinkTo' := 'TIID^Gerät 1 (EtherCAT)^Klemme 1 (EK1200)^Klemme 2 (EL3443)^L1 Status^Overvoltage'}
	MDP5001_341_L1_Status_Overvoltage			AT%I*  : BOOL;  // linked via attribute 
	{attribute 'TcLinkTo' := 'TIID^Gerät 1 (EtherCAT)^Klemme 1 (EK1200)^Klemme 2 (EL3443)^L1 Status^Overcurrent'}
	MDP5001_341_L1_Status_Overcurrent			AT%I*  : BOOL;  // linked via attribute 
	{attribute 'TcLinkTo' := 'TIID^Gerät 1 (EtherCAT)^Klemme 1 (EK1200)^Klemme 2 (EL3443)^L1 Status^Inaccurate Voltage'}	
	MDP5001_341_L1_Status_Inaccurate_Voltage	AT%I*  : BOOL;  // linked via attribute 
	{attribute 'TcLinkTo' := 'TIID^Gerät 1 (EtherCAT)^Klemme 1 (EK1200)^Klemme 2 (EL3443)^L1 Status^Inaccurate Current'}
	MDP5001_341_L1_Status_Inaccurate_Current	AT%I*  : BOOL;  // linked via attribute 	
	{attribute 'TcLinkTo' := 'TIID^Gerät 1 (EtherCAT)^Klemme 1 (EK1200)^Klemme 2 (EL3443)^L1 Status^Voltage Guard Warning'}
	MDP5001_341_L1_Status_Voltage_Guard_Warning	AT%I*  : BOOL;  // linked via attribute
	{attribute 'TcLinkTo' := 'TIID^Gerät 1 (EtherCAT)^Klemme 1 (EK1200)^Klemme 2 (EL3443)^L1 Status^Voltage Guard Error'}
	MDP5001_341_L1_Status_Voltage_Guard_Error	AT%I*  : BOOL;  // linked via attribute
	{attribute 'TcLinkTo' := 'TIID^Gerät 1 (EtherCAT)^Klemme 1 (EK1200)^Klemme 2 (EL3443)^L1 Status^Current Guard Warning'}
	MDP5001_341_L1_Status_Current_Guard_Warning AT%I*  : BOOL;  // linked via attribute
	{attribute 'TcLinkTo' := 'TIID^Gerät 1 (EtherCAT)^Klemme 1 (EK1200)^Klemme 2 (EL3443)^L1 Status^Current Guard Error'}
	MDP5001_341_L1_Status_Current_Guard_Error	AT%I*  : BOOL;  // linked via attribute
	{attribute 'TcLinkTo' := 'TIID^Gerät 1 (EtherCAT)^Klemme 1 (EK1200)^Klemme 2 (EL3443)^L1 Status^TxPDO Toggle'}
	MDP5001_341_L1_Status_TxPDO_Toggle			AT%I*  : BOOL;  // linked via attribute
	{attribute 'TcLinkTo' := 'TIID^Gerät 1 (EtherCAT)^Klemme 1 (EK1200)^Klemme 2 (EL3443)^L1 Basic^Voltage'}
	MDP5001_341_L1_Basic_Voltage				AT%I*  : REAL;		// linked via attribute 
	{attribute 'TcLinkTo' := 'TIID^Gerät 1 (EtherCAT)^Klemme 1 (EK1200)^Klemme 2 (EL3443)^L1 Basic^Current'}
	MDP5001_341_L1_Basic_Current				AT%I*  : REAL;		// linked via attribute 
	{attribute 'TcLinkTo' := 'TIID^Gerät 1 (EtherCAT)^Klemme 1 (EK1200)^Klemme 2 (EL3443)^L1 Power^Active Power'}
	MDP5001_341_L1_Power_Active_Power			AT%I*  : REAL;		// linked via attribute 
	{attribute 'TcLinkTo' := 'TIID^Gerät 1 (EtherCAT)^Klemme 1 (EK1200)^Klemme 2 (EL3443)^L1 Power^Apparent Power'}
	MDP5001_341_L1_Power_Apparent_Power			AT%I* : REAL;		// linked via attribute 
	{attribute 'TcLinkTo' := 'TIID^Gerät 1 (EtherCAT)^Klemme 1 (EK1200)^Klemme 2 (EL3443)^L1 Power^Reactive Power'}
	MDP5001_341_L1_Power_Reactive_Power			AT%I* : REAL;		// linked via attribute 
	{attribute 'TcLinkTo' := 'TIID^Gerät 1 (EtherCAT)^Klemme 1 (EK1200)^Klemme 2 (EL3443)^L1 Power^Power Factor'}
	MDP5001_341_L1_Power_Power_Factor			AT%I* : REAL;		// linked via attribute 
	{attribute 'TcLinkTo' := 'TIID^Gerät 1 (EtherCAT)^Klemme 1 (EK1200)^Klemme 2 (EL3443)^L2 Status^Voltage Sign Bit'}
	MDP5001_341_L2_Status_Voltage_Sign_Bit   	AT%I*  : BOOL;  // linked via attribute 
	{attribute 'TcLinkTo' := 'TIID^Gerät 1 (EtherCAT)^Klemme 1 (EK1200)^Klemme 2 (EL3443)^L2 Status^Overvoltage'}
	MDP5001_341_L2_Status_Overvoltage			AT%I*  : BOOL;  // linked via attribute 
	{attribute 'TcLinkTo' := 'TIID^Gerät 1 (EtherCAT)^Klemme 1 (EK1200)^Klemme 2 (EL3443)^L2 Status^Overcurrent'}
	MDP5001_341_L2_Status_Overcurrent			AT%I*  : BOOL;  // linked via attribute 
	{attribute 'TcLinkTo' := 'TIID^Gerät 1 (EtherCAT)^Klemme 1 (EK1200)^Klemme 2 (EL3443)^L2 Status^Inaccurate Voltage'}	
	MDP5001_341_L2_Status_Inaccurate_Voltage	AT%I*  : BOOL;  // linked via attribute 
	{attribute 'TcLinkTo' := 'TIID^Gerät 1 (EtherCAT)^Klemme 1 (EK1200)^Klemme 2 (EL3443)^L2 Status^Inaccurate Current'}
	MDP5001_341_L2_Status_Inaccurate_Current	AT%I*  : BOOL;  // linked via attribute 	
	{attribute 'TcLinkTo' := 'TIID^Gerät 1 (EtherCAT)^Klemme 1 (EK1200)^Klemme 2 (EL3443)^L2 Status^Voltage Guard Warning'}
	MDP5001_341_L2_Status_Voltage_Guard_Warning	AT%I*  : BOOL;  // linked via attribute
	{attribute 'TcLinkTo' := 'TIID^Gerät 1 (EtherCAT)^Klemme 1 (EK1200)^Klemme 2 (EL3443)^L2 Status^Voltage Guard Error'}
	MDP5001_341_L2_Status_Voltage_Guard_Error	AT%I*  : BOOL;  // linked via attribute
	{attribute 'TcLinkTo' := 'TIID^Gerät 1 (EtherCAT)^Klemme 1 (EK1200)^Klemme 2 (EL3443)^L2 Status^Current Guard Warning'}
	MDP5001_341_L2_Status_Current_Guard_Warning AT%I*  : BOOL;  // linked via attribute
	{attribute 'TcLinkTo' := 'TIID^Gerät 1 (EtherCAT)^Klemme 1 (EK1200)^Klemme 2 (EL3443)^L2 Status^Current Guard Error'}
	MDP5001_341_L2_Status_Current_Guard_Error	AT%I*  : BOOL;  // linked via attribute
	{attribute 'TcLinkTo' := 'TIID^Gerät 1 (EtherCAT)^Klemme 1 (EK1200)^Klemme 2 (EL3443)^L2 Status^TxPDO Toggle'}
	MDP5001_341_L2_Status_TxPDO_Toggle			AT%I*  : BOOL;  // linked via attribute
	{attribute 'TcLinkTo' := 'TIID^Gerät 1 (EtherCAT)^Klemme 1 (EK1200)^Klemme 2 (EL3443)^L2 Basic^Voltage'}
	MDP5001_341_L2_Basic_Voltage				AT%I* : REAL;		// linked via attribute 
	{attribute 'TcLinkTo' := 'TIID^Gerät 1 (EtherCAT)^Klemme 1 (EK1200)^Klemme 2 (EL3443)^L2 Basic^Current'}
	MDP5001_341_L2_Basic_Current				AT%I* : REAL;		// linked via attribute 
	{attribute 'TcLinkTo' := 'TIID^Gerät 1 (EtherCAT)^Klemme 1 (EK1200)^Klemme 2 (EL3443)^L2 Power^Active Power'}
	MDP5001_341_L2_Power_Active_Power			AT%I* : REAL;		// linked via attribute 
	{attribute 'TcLinkTo' := 'TIID^Gerät 1 (EtherCAT)^Klemme 1 (EK1200)^Klemme 2 (EL3443)^L2 Power^Apparent Power'}
	MDP5001_341_L2_Power_Apparent_Power			AT%I* : REAL;		// linked via attribute 
	{attribute 'TcLinkTo' := 'TIID^Gerät 1 (EtherCAT)^Klemme 1 (EK1200)^Klemme 2 (EL3443)^L2 Power^Reactive Power'}
	MDP5001_341_L2_Power_Reactive_Power			AT%I* : REAL;		// linked via attribute 
	{attribute 'TcLinkTo' := 'TIID^Gerät 1 (EtherCAT)^Klemme 1 (EK1200)^Klemme 2 (EL3443)^L2 Power^Power Factor'}
	MDP5001_341_L2_Power_Power_Factor			AT%I* : REAL;		// linked via attribute 
	{attribute 'TcLinkTo' := 'TIID^Gerät 1 (EtherCAT)^Klemme 1 (EK1200)^Klemme 2 (EL3443)^L3 Status^Voltage Sign Bit'}
	MDP5001_341_L3_Status_Voltage_Sign_Bit   	AT%I*  : BOOL;  // linked via attribute 
	{attribute 'TcLinkTo' := 'TIID^Gerät 1 (EtherCAT)^Klemme 1 (EK1200)^Klemme 2 (EL3443)^L3 Status^Overvoltage'}
	MDP5001_341_L3_Status_Overvoltage			AT%I*  : BOOL;  // linked via attribute 
	{attribute 'TcLinkTo' := 'TIID^Gerät 1 (EtherCAT)^Klemme 1 (EK1200)^Klemme 2 (EL3443)^L3 Status^Overcurrent'}
	MDP5001_341_L3_Status_Overcurrent			AT%I*  : BOOL;  // linked via attribute 
	{attribute 'TcLinkTo' := 'TIID^Gerät 1 (EtherCAT)^Klemme 1 (EK1200)^Klemme 2 (EL3443)^L3 Status^Inaccurate Voltage'}	
	MDP5001_341_L3_Status_Inaccurate_Voltage	AT%I*  : BOOL;  // linked via attribute 
	{attribute 'TcLinkTo' := 'TIID^Gerät 1 (EtherCAT)^Klemme 1 (EK1200)^Klemme 2 (EL3443)^L3 Status^Inaccurate Current'}
	MDP5001_341_L3_Status_Inaccurate_Current	AT%I*  : BOOL;  // linked via attribute 	
	{attribute 'TcLinkTo' := 'TIID^Gerät 1 (EtherCAT)^Klemme 1 (EK1200)^Klemme 2 (EL3443)^L3 Status^Voltage Guard Warning'}
	MDP5001_341_L3_Status_Voltage_Guard_Warning	AT%I*  : BOOL;  // linked via attribute
	{attribute 'TcLinkTo' := 'TIID^Gerät 1 (EtherCAT)^Klemme 1 (EK1200)^Klemme 2 (EL3443)^L3 Status^Voltage Guard Error'}
	MDP5001_341_L3_Status_Voltage_Guard_Error	AT%I*  : BOOL;  // linked via attribute
	{attribute 'TcLinkTo' := 'TIID^Gerät 1 (EtherCAT)^Klemme 1 (EK1200)^Klemme 2 (EL3443)^L3 Status^Current Guard Warning'}
	MDP5001_341_L3_Status_Current_Guard_Warning AT%I*  : BOOL;  // linked via attribute
	{attribute 'TcLinkTo' := 'TIID^Gerät 1 (EtherCAT)^Klemme 1 (EK1200)^Klemme 2 (EL3443)^L3 Status^Current Guard Error'}
	MDP5001_341_L3_Status_Current_Guard_Error	AT%I*  : BOOL;  // linked via attribute
	{attribute 'TcLinkTo' := 'TIID^Gerät 1 (EtherCAT)^Klemme 1 (EK1200)^Klemme 2 (EL3443)^L3 Status^TxPDO Toggle'}
	MDP5001_341_L3_Status_TxPDO_Toggle			AT%I*  : BOOL;  // linked via attribute
	{attribute 'TcLinkTo' := 'TIID^Gerät 1 (EtherCAT)^Klemme 1 (EK1200)^Klemme 2 (EL3443)^L3 Basic^Voltage'}
	MDP5001_341_L3_Basic_Voltage				AT%I* : REAL;		// linked via attribute 
	{attribute 'TcLinkTo' := 'TIID^Gerät 1 (EtherCAT)^Klemme 1 (EK1200)^Klemme 2 (EL3443)^L3 Basic^Current'}
	MDP5001_341_L3_Basic_Current				AT%I* : REAL;		// linked via attribute 
	{attribute 'TcLinkTo' := 'TIID^Gerät 1 (EtherCAT)^Klemme 1 (EK1200)^Klemme 2 (EL3443)^L3 Power^Active Power'}
	MDP5001_341_L3_Power_Active_Power			AT%I* : REAL;		// linked via attribute 
	{attribute 'TcLinkTo' := 'TIID^Gerät 1 (EtherCAT)^Klemme 1 (EK1200)^Klemme 2 (EL3443)^L3 Power^Apparent Power'}
	MDP5001_341_L3_Power_Apparent_Power			AT%I* : REAL;		// linked via attribute 
	{attribute 'TcLinkTo' := 'TIID^Gerät 1 (EtherCAT)^Klemme 1 (EK1200)^Klemme 2 (EL3443)^L3 Power^Reactive Power'}
	MDP5001_341_L3_Power_Reactive_Power			AT%I* : REAL;		// linked via attribute 
	{attribute 'TcLinkTo' := 'TIID^Gerät 1 (EtherCAT)^Klemme 1 (EK1200)^Klemme 2 (EL3443)^L3 Power^Power Factor'}
	MDP5001_341_L3_Power_Power_Factor			AT%I* : REAL;		// linked via attribute 
	{attribute 'TcLinkTo' := 'TIID^Gerät 1 (EtherCAT)^Klemme 1 (EK1200)^Klemme 2 (EL3443)^Total Status^System State'}
	MDP5001_341_Total_Status_System_State				AT%I* : BOOL;		// linked via attribute 
	{attribute 'TcLinkTo' := 'TIID^Gerät 1 (EtherCAT)^Klemme 1 (EK1200)^Klemme 2 (EL3443)^Total Status^Grid Direction'}
	MDP5001_341_Total_Status_Grid_Direction				AT%I* : BOOL;		// linked via attribute 
	{attribute 'TcLinkTo' := 'TIID^Gerät 1 (EtherCAT)^Klemme 1 (EK1200)^Klemme 2 (EL3443)^Total Status^Frequency Guard Warning'}
	MDP5001_341_Total_Status_Frequency_Guard_Warning	AT%I* : BOOL;		// linked via attribute 
	{attribute 'TcLinkTo' := 'TIID^Gerät 1 (EtherCAT)^Klemme 1 (EK1200)^Klemme 2 (EL3443)^Total Status^Frequency Guard Error'}
	MDP5001_341_Total_Status_Frequency_Guard_Error		AT%I* : BOOL;		// linked via attribute 
	{attribute 'TcLinkTo' := 'TIID^Gerät 1 (EtherCAT)^Klemme 1 (EK1200)^Klemme 2 (EL3443)^Total Status^Neutral Current Guard Warning'}
	MDP5001_341_Total_Status_Neutral_Current_Guard_Warning	AT%I* : BOOL;		// linked via attribute 
	{attribute 'TcLinkTo' := 'TIID^Gerät 1 (EtherCAT)^Klemme 1 (EK1200)^Klemme 2 (EL3443)^Total Status^Neutral Current Guard Error'}
	MDP5001_341_Total_Status_Neutral_Current_Guard_Error	AT%I* : BOOL;		// linked via attribute 
	{attribute 'TcLinkTo' := 'TIID^Gerät 1 (EtherCAT)^Klemme 1 (EK1200)^Klemme 2 (EL3443)^Total Status^Active Power Guard Warning'}
	MDP5001_341_Total_Status_Active_Power_Guard_Warning		AT%I* : BOOL;		// linked via attribute 
	{attribute 'TcLinkTo' := 'TIID^Gerät 1 (EtherCAT)^Klemme 1 (EK1200)^Klemme 2 (EL3443)^Total Status^Active Power Guard Error'}
	MDP5001_341_Total_Status_Active_Power_Guard_Error		AT%I* : BOOL;		// linked via attribute 
	{attribute 'TcLinkTo' := 'TIID^Gerät 1 (EtherCAT)^Klemme 1 (EK1200)^Klemme 2 (EL3443)^Total Status^Apparent Power Guard Warning'}
	MDP5001_341_Total_Status_Apparent_Power_Guard_Warning	AT%I* : BOOL;		// linked via attribute 
	{attribute 'TcLinkTo' := 'TIID^Gerät 1 (EtherCAT)^Klemme 1 (EK1200)^Klemme 2 (EL3443)^Total Status^Apparent Power Guard Error'}
	MDP5001_341_Total_Status_Apparent_Power_Guard_Error		AT%I* : BOOL;		// linked via attribute 
	{attribute 'TcLinkTo' := 'TIID^Gerät 1 (EtherCAT)^Klemme 1 (EK1200)^Klemme 2 (EL3443)^Total Status^Power Quality Guard Warning'}
	MDP5001_341_Total_Status_Power_Quality_Guard_Warning	AT%I* : BOOL;		// linked via attribute 
	{attribute 'TcLinkTo' := 'TIID^Gerät 1 (EtherCAT)^Klemme 1 (EK1200)^Klemme 2 (EL3443)^Total Status^Power Quality Guard Error'}
	MDP5001_341_Total_Status_Power_Quality_Guard_Error		AT%I* : BOOL;		// linked via attribute 
	{attribute 'TcLinkTo' := 'TIID^Gerät 1 (EtherCAT)^Klemme 1 (EK1200)^Klemme 2 (EL3443)^Total Status^TxPDO State'}
	MDP5001_341_Total_Status_TxPDO_State					AT%I* : BOOL;		// linked via attribute 
	{attribute 'TcLinkTo' := 'TIID^Gerät 1 (EtherCAT)^Klemme 1 (EK1200)^Klemme 2 (EL3443)^Total Status^TxPDO Toggle'}
	MDP5001_341_Total_Status_TxPDO_Toggle					AT%I* : BOOL;		// linked via attribute 
	{attribute 'TcLinkTo' := 'TIID^Gerät 1 (EtherCAT)^Klemme 1 (EK1200)^Klemme 2 (EL3443)^Total Status^Power Quality Factor'}
	MDP5001_341_Total_Status_Power_Quality_Factor			AT%I* : REAL;		// linked via attribute 
	{attribute 'TcLinkTo' := 'TIID^Gerät 1 (EtherCAT)^Klemme 1 (EK1200)^Klemme 2 (EL3443)^Total Basic^Frequency'}
	MDP5001_341_Total_Basic_Frequency						AT%I* : REAL;		// linked via attribute 
	{attribute 'TcLinkTo' := 'TIID^Gerät 1 (EtherCAT)^Klemme 1 (EK1200)^Klemme 2 (EL3443)^Total Basic^Power Factor'}
	MDP5001_341_Total_Basic_Power_Factor					AT%I* : REAL;		// linked via attribute 
	{attribute 'TcLinkTo' := 'TIID^Gerät 1 (EtherCAT)^Klemme 1 (EK1200)^Klemme 2 (EL3443)^Total Basic^Calculated Neutral Line Current'}
	MDP5001_341_Total_Basic_Calculated_Neutral_Line_Current	AT%I* : REAL;		// linked via attribute 
	{attribute 'TcLinkTo' := 'TIID^Gerät 1 (EtherCAT)^Klemme 1 (EK1200)^Klemme 2 (EL3443)^Total Variant Value In^TxPDO Toggle'}
	MDP5001_341_Total_Variant_Value_In_TxPDO_Toggle			AT%I* : BOOL;		// linked via attribute 
	{attribute 'TcLinkTo' := 'TIID^Gerät 1 (EtherCAT)^Klemme 1 (EK1200)^Klemme 2 (EL3443)^Total Variant Value In^Index 1 REAL'}
	MDP5001_341_Total_Variant_Value_In_Index_1_REAL			AT%I* : UINT;		// linked via attribute 
	{attribute 'TcLinkTo' := 'TIID^Gerät 1 (EtherCAT)^Klemme 1 (EK1200)^Klemme 2 (EL3443)^Total Variant Value In^Value 1 REAL'}
	MDP5001_341_Total_Variant_Value_In_Value_1_REAL			AT%I* : REAL;		// linked via attribute 
	{attribute 'TcLinkTo' := 'TIID^Gerät 1 (EtherCAT)^Klemme 1 (EK1200)^Klemme 2 (EL3443)^Total Variant Value In^Index 2 REAL'}
	MDP5001_341_Total_Variant_Value_In_Index_2_REAL			AT%I* : UINT;		// linked via attribute 
	{attribute 'TcLinkTo' := 'TIID^Gerät 1 (EtherCAT)^Klemme 1 (EK1200)^Klemme 2 (EL3443)^Total Variant Value In^Value 2 REAL'}
	MDP5001_341_Total_Variant_Value_In_Value_2_REAL			AT%I* : REAL;		// linked via attribute 
	{attribute 'TcLinkTo' := 'TIID^Gerät 1 (EtherCAT)^Klemme 1 (EK1200)^Klemme 2 (EL3443)^Total Variant Value In^Index 3 REAL'}
	MDP5001_341_Total_Variant_Value_In_Index_3_REAL			AT%I* : UINT;		// linked via attribute 
	{attribute 'TcLinkTo' := 'TIID^Gerät 1 (EtherCAT)^Klemme 1 (EK1200)^Klemme 2 (EL3443)^Total Variant Value In^Value 3 REAL'}
	MDP5001_341_Total_Variant_Value_In_Value_3_REAL			AT%I* : REAL;		// linked via attribute 
	{attribute 'TcLinkTo' := 'TIID^Gerät 1 (EtherCAT)^Klemme 1 (EK1200)^Klemme 2 (EL3443)^Total Variant Value In^Index 4 ULINT'}
	MDP5001_341_Total_Variant_Value_In_Index_4_ULINT		AT%I* : UINT;		// linked via attribute 
	{attribute 'TcLinkTo' := 'TIID^Gerät 1 (EtherCAT)^Klemme 1 (EK1200)^Klemme 2 (EL3443)^Total Variant Value In^Value 4 ULINT'}
	MDP5001_341_Total_Variant_Value_In_Value_4_ULINT		AT%I* : ULINT;	// linked via attribute 
	{attribute 'TcLinkTo' := 'TIID^Gerät 1 (EtherCAT)^Klemme 1 (EK1200)^Klemme 2 (EL3443)^DPM Data^Data 1'}
	MDP5001_341_DPM_Data_Data_1								AT%I* : UDINT;	// linked via attribute 
	{attribute 'TcLinkTo' := 'TIID^Gerät 1 (EtherCAT)^Klemme 1 (EK1200)^Klemme 2 (EL3443)^DPM Data^Data 2'}
	MDP5001_341_DPM_Data_Data_2								AT%I* : UDINT;	// linked via attribute 
	{attribute 'TcLinkTo' := 'TIID^Gerät 1 (EtherCAT)^Klemme 1 (EK1200)^Klemme 2 (EL3443)^DPM Data^Data 3'}
	MDP5001_341_DPM_Data_Data_3								AT%I* : UDINT;	// linked via attribute 
	{attribute 'TcLinkTo' := 'TIID^Gerät 1 (EtherCAT)^Klemme 1 (EK1200)^Klemme 2 (EL3443)^DPM Data^Data 4'}
	MDP5001_341_DPM_Data_Data_4								AT%I* : UDINT;	// linked via attribute 
	{attribute 'TcLinkTo' := 'TIID^Gerät 1 (EtherCAT)^Klemme 1 (EK1200)^Klemme 2 (EL3443)^DPM Data^Data 5'}
	MDP5001_341_DPM_Data_Data_5								AT%I* : UDINT;	// linked via attribute 
	{attribute 'TcLinkTo' := 'TIID^Gerät 1 (EtherCAT)^Klemme 1 (EK1200)^Klemme 2 (EL3443)^DPM Data^Data 6'}
	MDP5001_341_DPM_Data_Data_6								AT%I* : UDINT;	// linked via attribute 
	{attribute 'TcLinkTo' := 'TIID^Gerät 1 (EtherCAT)^Klemme 1 (EK1200)^Klemme 2 (EL3443)^DPM Data^Data 7'}
	MDP5001_341_DPM_Data_Data_7								AT%I* : UDINT;	// linked via attribute 
	{attribute 'TcLinkTo' := 'TIID^Gerät 1 (EtherCAT)^Klemme 1 (EK1200)^Klemme 2 (EL3443)^DPM Data^Data 8'}
	MDP5001_341_DPM_Data_Data_8								AT%I* : UDINT;	// linked via attribute 
	{attribute 'TcLinkTo' := 'TIID^Gerät 1 (EtherCAT)^Klemme 1 (EK1200)^Klemme 2 (EL3443)^DPM Data^Data 9'}
	MDP5001_341_DPM_Data_Data_9								AT%I* : UDINT;	// linked via attribute 
	{attribute 'TcLinkTo' := 'TIID^Gerät 1 (EtherCAT)^Klemme 1 (EK1200)^Klemme 2 (EL3443)^DPM Data^Data 10'}
	MDP5001_341_DPM_Data_Data_10							AT%I* : UDINT;	// linked via attribute 
	{attribute 'TcLinkTo' := 'TIID^Gerät 1 (EtherCAT)^Klemme 1 (EK1200)^Klemme 2 (EL3443)^DPM Data^Data 11'}
	MDP5001_341_DPM_Data_Data_11							AT%I* : UDINT;	// linked via attribute 
	{attribute 'TcLinkTo' := 'TIID^Gerät 1 (EtherCAT)^Klemme 1 (EK1200)^Klemme 2 (EL3443)^DPM Data^Data 12'}
	MDP5001_341_DPM_Data_Data_12							AT%I* : UDINT;	// linked via attribute 
	{attribute 'TcLinkTo' := 'TIID^Gerät 1 (EtherCAT)^Klemme 1 (EK1200)^Klemme 2 (EL3443)^DPM Data^Data 13'}
	MDP5001_341_DPM_Data_Data_13							AT%I* : UDINT;	// linked via attribute 
	{attribute 'TcLinkTo' := 'TIID^Gerät 1 (EtherCAT)^Klemme 1 (EK1200)^Klemme 2 (EL3443)^DPM Data^Data 14'}
	MDP5001_341_DPM_Data_Data_14							AT%I* : UDINT;	// linked via attribute 
	{attribute 'TcLinkTo' := 'TIID^Gerät 1 (EtherCAT)^Klemme 1 (EK1200)^Klemme 2 (EL3443)^DPM Data^Data 15'}
	MDP5001_341_DPM_Data_Data_15							AT%I* : UDINT;	// linked via attribute 
	{attribute 'TcLinkTo' := 'TIID^Gerät 1 (EtherCAT)^Klemme 1 (EK1200)^Klemme 2 (EL3443)^DPM Data^Data 16'}
	MDP5001_341_DPM_Data_Data_16							AT%I* : UDINT;	// linked via attribute 
	{attribute 'TcLinkTo' := 'TIID^Gerät 1 (EtherCAT)^Klemme 1 (EK1200)^Klemme 2 (EL3443)^DPM Data^Data 17'}
	MDP5001_341_DPM_Data_Data_17							AT%I* : UDINT;	// linked via attribute 
	{attribute 'TcLinkTo' := 'TIID^Gerät 1 (EtherCAT)^Klemme 1 (EK1200)^Klemme 2 (EL3443)^DPM Data^Data 18'}
	MDP5001_341_DPM_Data_Data_18							AT%I* : UDINT;	// linked via attribute 
	{attribute 'TcLinkTo' := 'TIID^Gerät 1 (EtherCAT)^Klemme 1 (EK1200)^Klemme 2 (EL3443)^DPM Data^Data 19'}
	MDP5001_341_DPM_Data_Data_19							AT%I* : UDINT;	// linked via attribute 
	{attribute 'TcLinkTo' := 'TIID^Gerät 1 (EtherCAT)^Klemme 1 (EK1200)^Klemme 2 (EL3443)^DPM Data^Data 20'}
	MDP5001_341_DPM_Data_Data_20							AT%I* : UDINT;	// linked via attribute 
	{attribute 'TcLinkTo' := 'TIID^Gerät 1 (EtherCAT)^Klemme 1 (EK1200)^Klemme 2 (EL3443)^Total Variant Value Out^Index 1 REAL'}
	MDP5001_341_Total_Variant_Value_Out_Index_1_REAL	AT%Q* : UINT;
	{attribute 'TcLinkTo' := 'TIID^Gerät 1 (EtherCAT)^Klemme 1 (EK1200)^Klemme 2 (EL3443)^Total Variant Value Out^Index 2 REAL'}
	MDP5001_341_Total_Variant_Value_Out_Index_2_REAL	AT%Q* : UINT;
	{attribute 'TcLinkTo' := 'TIID^Gerät 1 (EtherCAT)^Klemme 1 (EK1200)^Klemme 2 (EL3443)^Total Variant Value Out^Index 3 REAL'}
	MDP5001_341_Total_Variant_Value_Out_Index_3_REAL	AT%Q* : UINT;
	{attribute 'TcLinkTo' := 'TIID^Gerät 1 (EtherCAT)^Klemme 1 (EK1200)^Klemme 2 (EL3443)^Total Variant Value Out^Index 4 ULINT'}
	MDP5001_341_Total_Variant_Value_Out_Index_4_ULINT	AT%Q* : UINT;
	{attribute 'TcLinkTo' := 'TIID^Gerät 1 (EtherCAT)^Klemme 1 (EK1200)^Klemme 2 (EL3443)^Total Interval^Reset Interval'}
	MDP5001_341_Total_Interval_Reset_Interval			AT%Q* : BOOL;
	
// IOs for EL3446
	{attribute 'TcLinkTo' := 'TIID^Gerät 1 (EtherCAT)^Klemme 1 (EK1200)^Klemme 3 (EL3446)^I1 Channel^Overcurrent'}
	MDP5001_342_I1_Channel_Overcurrent_1						AT%I*  : BOOL;
	{attribute 'TcLinkTo' := 'TIID^Gerät 1 (EtherCAT)^Klemme 1 (EK1200)^Klemme 3 (EL3446)^I1 Channel^Inaccurate Current'}
	MDP5001_342_I1_Channel_Inaccurate_Current_1				AT%I*  : BOOL;
	{attribute 'TcLinkTo' := 'TIID^Gerät 1 (EtherCAT)^Klemme 1 (EK1200)^Klemme 3 (EL3446)^I1 Channel^Current Guard Warning'}
	MDP5001_342_I1_Channel_Current_Guard_Warning_1			AT%I*  : bool;
	{attribute 'TcLinkTo' := 'TIID^Gerät 1 (EtherCAT)^Klemme 1 (EK1200)^Klemme 3 (EL3446)^I1 Channel^Current Guard Error'}
	MDP5001_342_I1_Channel_Current_Guard_Error_1				AT%I*  : bool;
	{attribute 'TcLinkTo' := 'TIID^Gerät 1 (EtherCAT)^Klemme 1 (EK1200)^Klemme 3 (EL3446)^I1 Channel^Apparent Power Guard Warning'}
	MDP5001_342_I1_Channel_Apparent_Power_Guard_Warning_1		AT%I*  : bool;
	{attribute 'TcLinkTo' := 'TIID^Gerät 1 (EtherCAT)^Klemme 1 (EK1200)^Klemme 3 (EL3446)^I1 Channel^Apparent Power Guard Error'}
	MDP5001_342_I1_Channel_Apparent_Power_Guard_Error_1		AT%I*  : bool;
	{attribute 'TcLinkTo' := 'TIID^Gerät 1 (EtherCAT)^Klemme 1 (EK1200)^Klemme 3 (EL3446)^I1 Channel^Active Power Guard Warning'}
	MDP5001_342_I1_Channel_Active_Power_Guard_Warning_1		AT%I*  : bool;
	{attribute 'TcLinkTo' := 'TIID^Gerät 1 (EtherCAT)^Klemme 1 (EK1200)^Klemme 3 (EL3446)^I1 Channel^Active Power Guard Error'}
	MDP5001_342_I1_Channel_Active_Power_Guard_Error_1			AT%I*  : bool;
	{attribute 'TcLinkTo' := 'TIID^Gerät 1 (EtherCAT)^Klemme 1 (EK1200)^Klemme 3 (EL3446)^I1 Channel^Reactive Power Guard Warning'}
	MDP5001_342_I1_Channel_Reactive_Power_Guard_Warning_1		AT%I*  : bool;
	{attribute 'TcLinkTo' := 'TIID^Gerät 1 (EtherCAT)^Klemme 1 (EK1200)^Klemme 3 (EL3446)^I1 Channel^Reactive Power Guard Error'}
	MDP5001_342_I1_Channel_Reactive_Power_Guard_Error_1		AT%I*  : bool;
	{attribute 'TcLinkTo' := 'TIID^Gerät 1 (EtherCAT)^Klemme 1 (EK1200)^Klemme 3 (EL3446)^I1 Channel^DPM Inaccurate'}
	MDP5001_342_I1_Channel_DPM_Inaccurate_1					AT%I*  : bool;
	{attribute 'TcLinkTo' := 'TIID^Gerät 1 (EtherCAT)^Klemme 1 (EK1200)^Klemme 3 (EL3446)^I1 Channel^DPM Timeout'}
	MDP5001_342_I1_Channel_DPM_Timeout_1						AT%I*  : bool;
	{attribute 'TcLinkTo' := 'TIID^Gerät 1 (EtherCAT)^Klemme 1 (EK1200)^Klemme 3 (EL3446)^I1 Channel^TxPDO Toggle'}
	MDP5001_342_I1_Channel_TxPDO_Toggle_1						AT%I*  : bool;
	{attribute 'TcLinkTo' := 'TIID^Gerät 1 (EtherCAT)^Klemme 1 (EK1200)^Klemme 3 (EL3446)^I1 Channel^Current'}
	MDP5001_342_I1_Channel_Current_1							AT%I*  : REAL;
	{attribute 'TcLinkTo' := 'TIID^Gerät 1 (EtherCAT)^Klemme 1 (EK1200)^Klemme 3 (EL3446)^I1 Channel^Active Power'}
	MDP5001_342_I1_Channel_Active_Power_1						AT%I*  : REAL;
	{attribute 'TcLinkTo' := 'TIID^Gerät 1 (EtherCAT)^Klemme 1 (EK1200)^Klemme 3 (EL3446)^I1 Channel^Apparent Power'}
	MDP5001_342_I1_Channel_Apparent_Power_1					AT%I*  : REAL;
	{attribute 'TcLinkTo' := 'TIID^Gerät 1 (EtherCAT)^Klemme 1 (EK1200)^Klemme 3 (EL3446)^I1 Channel^Reactive Power Fundamental'}
	MDP5001_342_I1_Channel_Reactive_Power_Fundamental_1		AT%I*  : REAL;
	{attribute 'TcLinkTo' := 'TIID^Gerät 1 (EtherCAT)^Klemme 1 (EK1200)^Klemme 3 (EL3446)^I1 Channel^Active Energy'}
	MDP5001_342_I1_Channel_Active_Energy_1					AT%I*  : DINT;
	{attribute 'TcLinkTo' := 'TIID^Gerät 1 (EtherCAT)^Klemme 1 (EK1200)^Klemme 3 (EL3446)^I2 Channel^Overcurrent'}
	MDP5001_342_I2_Channel_Overcurrent_1						AT%I*  : BOOL;
	{attribute 'TcLinkTo' := 'TIID^Gerät 1 (EtherCAT)^Klemme 1 (EK1200)^Klemme 3 (EL3446)^I2 Channel^Inaccurate Current'}
	MDP5001_342_I2_Channel_Inaccurate_Current_1				AT%I*  : BOOL;
	{attribute 'TcLinkTo' := 'TIID^Gerät 1 (EtherCAT)^Klemme 1 (EK1200)^Klemme 3 (EL3446)^I2 Channel^Current Guard Warning'}
	MDP5001_342_I2_Channel_Current_Guard_Warning_1			AT%I*  : bool;
	{attribute 'TcLinkTo' := 'TIID^Gerät 1 (EtherCAT)^Klemme 1 (EK1200)^Klemme 3 (EL3446)^I2 Channel^Current Guard Error'}
	MDP5001_342_I2_Channel_Current_Guard_Error_1				AT%I*  : bool;
	{attribute 'TcLinkTo' := 'TIID^Gerät 1 (EtherCAT)^Klemme 1 (EK1200)^Klemme 3 (EL3446)^I2 Channel^Apparent Power Guard Warning'}
	MDP5001_342_I2_Channel_Apparent_Power_Guard_Warning_1		AT%I*  : bool;
	{attribute 'TcLinkTo' := 'TIID^Gerät 1 (EtherCAT)^Klemme 1 (EK1200)^Klemme 3 (EL3446)^I2 Channel^Apparent Power Guard Error'}
	MDP5001_342_I2_Channel_Apparent_Power_Guard_Error_1		AT%I*  : bool;
	{attribute 'TcLinkTo' := 'TIID^Gerät 1 (EtherCAT)^Klemme 1 (EK1200)^Klemme 3 (EL3446)^I2 Channel^Active Power Guard Warning'}
	MDP5001_342_I2_Channel_Active_Power_Guard_Warning_1		AT%I*  : bool;
	{attribute 'TcLinkTo' := 'TIID^Gerät 1 (EtherCAT)^Klemme 1 (EK1200)^Klemme 3 (EL3446)^I2 Channel^Active Power Guard Error'}
	MDP5001_342_I2_Channel_Active_Power_Guard_Error_1			AT%I*  : bool;
	{attribute 'TcLinkTo' := 'TIID^Gerät 1 (EtherCAT)^Klemme 1 (EK1200)^Klemme 3 (EL3446)^I2 Channel^Reactive Power Guard Warning'}
	MDP5001_342_I2_Channel_Reactive_Power_Guard_Warning_1		AT%I*  : bool;
	{attribute 'TcLinkTo' := 'TIID^Gerät 1 (EtherCAT)^Klemme 1 (EK1200)^Klemme 3 (EL3446)^I2 Channel^Reactive Power Guard Error'}
	MDP5001_342_I2_Channel_Reactive_Power_Guard_Error_1		AT%I*  : bool;
	{attribute 'TcLinkTo' := 'TIID^Gerät 1 (EtherCAT)^Klemme 1 (EK1200)^Klemme 3 (EL3446)^I2 Channel^DPM Inaccurate'}
	MDP5001_342_I2_Channel_DPM_Inaccurate_1					AT%I*  : bool;
	{attribute 'TcLinkTo' := 'TIID^Gerät 1 (EtherCAT)^Klemme 1 (EK1200)^Klemme 3 (EL3446)^I2 Channel^DPM Timeout'}
	MDP5001_342_I2_Channel_DPM_Timeout_1						AT%I*  : bool;
	{attribute 'TcLinkTo' := 'TIID^Gerät 1 (EtherCAT)^Klemme 1 (EK1200)^Klemme 3 (EL3446)^I2 Channel^TxPDO Toggle'}
	MDP5001_342_I2_Channel_TxPDO_Toggle_1						AT%I*  : bool;
	{attribute 'TcLinkTo' := 'TIID^Gerät 1 (EtherCAT)^Klemme 1 (EK1200)^Klemme 3 (EL3446)^I2 Channel^Current'}
	MDP5001_342_I2_Channel_Current_1							AT%I*  : REAL;
	{attribute 'TcLinkTo' := 'TIID^Gerät 1 (EtherCAT)^Klemme 1 (EK1200)^Klemme 3 (EL3446)^I2 Channel^Active Power'}
	MDP5001_342_I2_Channel_Active_Power_1						AT%I*  : REAL;
	{attribute 'TcLinkTo' := 'TIID^Gerät 1 (EtherCAT)^Klemme 1 (EK1200)^Klemme 3 (EL3446)^I2 Channel^Apparent Power'}
	MDP5001_342_I2_Channel_Apparent_Power_1					AT%I*  : REAL;
	{attribute 'TcLinkTo' := 'TIID^Gerät 1 (EtherCAT)^Klemme 1 (EK1200)^Klemme 3 (EL3446)^I2 Channel^Reactive Power Fundamental'}
	MDP5001_342_I2_Channel_Reactive_Power_Fundamental_1		AT%I*  : REAL;
	{attribute 'TcLinkTo' := 'TIID^Gerät 1 (EtherCAT)^Klemme 1 (EK1200)^Klemme 3 (EL3446)^I2 Channel^Active Energy'}
	MDP5001_342_I2_Channel_Active_Energy_1					AT%I*  : DINT;
	{attribute 'TcLinkTo' := 'TIID^Gerät 1 (EtherCAT)^Klemme 1 (EK1200)^Klemme 3 (EL3446)^I3 Channel^Overcurrent'}
	MDP5001_342_I3_Channel_Overcurrent_1						AT%I*  : BOOL;
	{attribute 'TcLinkTo' := 'TIID^Gerät 1 (EtherCAT)^Klemme 1 (EK1200)^Klemme 3 (EL3446)^I3 Channel^Inaccurate Current'}
	MDP5001_342_I3_Channel_Inaccurate_Current_1				AT%I*  : BOOL;
	{attribute 'TcLinkTo' := 'TIID^Gerät 1 (EtherCAT)^Klemme 1 (EK1200)^Klemme 3 (EL3446)^I3 Channel^Current Guard Warning'}
	MDP5001_342_I3_Channel_Current_Guard_Warning_1			AT%I*  : bool;
	{attribute 'TcLinkTo' := 'TIID^Gerät 1 (EtherCAT)^Klemme 1 (EK1200)^Klemme 3 (EL3446)^I3 Channel^Current Guard Error'}
	MDP5001_342_I3_Channel_Current_Guard_Error_1				AT%I*  : bool;
	{attribute 'TcLinkTo' := 'TIID^Gerät 1 (EtherCAT)^Klemme 1 (EK1200)^Klemme 3 (EL3446)^I3 Channel^Apparent Power Guard Warning'}
	MDP5001_342_I3_Channel_Apparent_Power_Guard_Warning_1		AT%I*  : bool;
	{attribute 'TcLinkTo' := 'TIID^Gerät 1 (EtherCAT)^Klemme 1 (EK1200)^Klemme 3 (EL3446)^I3 Channel^Apparent Power Guard Error'}
	MDP5001_342_I3_Channel_Apparent_Power_Guard_Error_1		AT%I*  : bool;
	{attribute 'TcLinkTo' := 'TIID^Gerät 1 (EtherCAT)^Klemme 1 (EK1200)^Klemme 3 (EL3446)^I3 Channel^Active Power Guard Warning'}
	MDP5001_342_I3_Channel_Active_Power_Guard_Warning_1		AT%I*  : bool;
	{attribute 'TcLinkTo' := 'TIID^Gerät 1 (EtherCAT)^Klemme 1 (EK1200)^Klemme 3 (EL3446)^I3 Channel^Active Power Guard Error'}
	MDP5001_342_I3_Channel_Active_Power_Guard_Error_1		AT%I*  : bool;
	{attribute 'TcLinkTo' := 'TIID^Gerät 1 (EtherCAT)^Klemme 1 (EK1200)^Klemme 3 (EL3446)^I3 Channel^Reactive Power Guard Warning'}
	MDP5001_342_I3_Channel_Reactive_Power_Guard_Warning_1		AT%I*  : bool;
	{attribute 'TcLinkTo' := 'TIID^Gerät 1 (EtherCAT)^Klemme 1 (EK1200)^Klemme 3 (EL3446)^I3 Channel^Reactive Power Guard Error'}
	MDP5001_342_I3_Channel_Reactive_Power_Guard_Error_1		AT%I*  : bool;
	{attribute 'TcLinkTo' := 'TIID^Gerät 1 (EtherCAT)^Klemme 1 (EK1200)^Klemme 3 (EL3446)^I3 Channel^DPM Inaccurate'}
	MDP5001_342_I3_Channel_DPM_Inaccurate_1					AT%I*  : bool;
	{attribute 'TcLinkTo' := 'TIID^Gerät 1 (EtherCAT)^Klemme 1 (EK1200)^Klemme 3 (EL3446)^I3 Channel^DPM Timeout'}
	MDP5001_342_I3_Channel_DPM_Timeout_1						AT%I*  : bool;
	{attribute 'TcLinkTo' := 'TIID^Gerät 1 (EtherCAT)^Klemme 1 (EK1200)^Klemme 3 (EL3446)^I3 Channel^TxPDO Toggle'}
	MDP5001_342_I3_Channel_TxPDO_Toggle_1						AT%I*  : bool;
	{attribute 'TcLinkTo' := 'TIID^Gerät 1 (EtherCAT)^Klemme 1 (EK1200)^Klemme 3 (EL3446)^I3 Channel^Current'}
	MDP5001_342_I3_Channel_Current_1							AT%I*  : REAL;
	{attribute 'TcLinkTo' := 'TIID^Gerät 1 (EtherCAT)^Klemme 1 (EK1200)^Klemme 3 (EL3446)^I3 Channel^Active Power'}
	MDP5001_342_I3_Channel_Active_Power_1						AT%I*  : REAL;
	{attribute 'TcLinkTo' := 'TIID^Gerät 1 (EtherCAT)^Klemme 1 (EK1200)^Klemme 3 (EL3446)^I3 Channel^Apparent Power'}
	MDP5001_342_I3_Channel_Apparent_Power_1					AT%I*  : REAL;
	{attribute 'TcLinkTo' := 'TIID^Gerät 1 (EtherCAT)^Klemme 1 (EK1200)^Klemme 3 (EL3446)^I3 Channel^Reactive Power Fundamental'}
	MDP5001_342_I3_Channel_Reactive_Power_Fundamental_1		AT%I*  : REAL;
	{attribute 'TcLinkTo' := 'TIID^Gerät 1 (EtherCAT)^Klemme 1 (EK1200)^Klemme 3 (EL3446)^I3 Channel^Active Energy'}
	MDP5001_342_I3_Channel_Active_Energy_1					AT%I*  : DINT;	
	{attribute 'TcLinkTo' := 'TIID^Gerät 1 (EtherCAT)^Klemme 1 (EK1200)^Klemme 3 (EL3446)^I4 Channel^Overcurrent'}
	MDP5001_342_I4_Channel_Overcurrent_1						AT%I*  : BOOL;
	{attribute 'TcLinkTo' := 'TIID^Gerät 1 (EtherCAT)^Klemme 1 (EK1200)^Klemme 3 (EL3446)^I4 Channel^Inaccurate Current'}
	MDP5001_342_I4_Channel_Inaccurate_Current_1				AT%I*  : BOOL;
	{attribute 'TcLinkTo' := 'TIID^Gerät 1 (EtherCAT)^Klemme 1 (EK1200)^Klemme 3 (EL3446)^I4 Channel^Current Guard Warning'}
	MDP5001_342_I4_Channel_Current_Guard_Warning_1			AT%I*  : bool;
	{attribute 'TcLinkTo' := 'TIID^Gerät 1 (EtherCAT)^Klemme 1 (EK1200)^Klemme 3 (EL3446)^I4 Channel^Current Guard Error'}
	MDP5001_342_I4_Channel_Current_Guard_Error_1				AT%I*  : bool;
	{attribute 'TcLinkTo' := 'TIID^Gerät 1 (EtherCAT)^Klemme 1 (EK1200)^Klemme 3 (EL3446)^I4 Channel^Apparent Power Guard Warning'}
	MDP5001_342_I4_Channel_Apparent_Power_Guard_Warning_1		AT%I*  : bool;
	{attribute 'TcLinkTo' := 'TIID^Gerät 1 (EtherCAT)^Klemme 1 (EK1200)^Klemme 3 (EL3446)^I4 Channel^Apparent Power Guard Error'}
	MDP5001_342_I4_Channel_Apparent_Power_Guard_Error_1		AT%I*  : bool;
	{attribute 'TcLinkTo' := 'TIID^Gerät 1 (EtherCAT)^Klemme 1 (EK1200)^Klemme 3 (EL3446)^I4 Channel^Active Power Guard Warning'}
	MDP5001_342_I4_Channel_Active_Power_Guard_Warning_1		AT%I*  : bool;
	{attribute 'TcLinkTo' := 'TIID^Gerät 1 (EtherCAT)^Klemme 1 (EK1200)^Klemme 3 (EL3446)^I4 Channel^Active Power Guard Error'}
	MDP5001_342_I4_Channel_Active_Power_Guard_Error_1			AT%I*  : bool;
	{attribute 'TcLinkTo' := 'TIID^Gerät 1 (EtherCAT)^Klemme 1 (EK1200)^Klemme 3 (EL3446)^I4 Channel^Reactive Power Guard Warning'}
	MDP5001_342_I4_Channel_Reactive_Power_Guard_Warning_1		AT%I*  : bool;
	{attribute 'TcLinkTo' := 'TIID^Gerät 1 (EtherCAT)^Klemme 1 (EK1200)^Klemme 3 (EL3446)^I4 Channel^Reactive Power Guard Error'}
	MDP5001_342_I4_Channel_Reactive_Power_Guard_Error_1		AT%I*  : bool;
	{attribute 'TcLinkTo' := 'TIID^Gerät 1 (EtherCAT)^Klemme 1 (EK1200)^Klemme 3 (EL3446)^I4 Channel^DPM Inaccurate'}
	MDP5001_342_I4_Channel_DPM_Inaccurate_1					AT%I*  : bool;
	{attribute 'TcLinkTo' := 'TIID^Gerät 1 (EtherCAT)^Klemme 1 (EK1200)^Klemme 3 (EL3446)^I4 Channel^DPM Timeout'}
	MDP5001_342_I4_Channel_DPM_Timeout_1						AT%I*  : bool;
	{attribute 'TcLinkTo' := 'TIID^Gerät 1 (EtherCAT)^Klemme 1 (EK1200)^Klemme 3 (EL3446)^I4 Channel^TxPDO Toggle'}
	MDP5001_342_I4_Channel_TxPDO_Toggle_1						AT%I*  : bool;
	{attribute 'TcLinkTo' := 'TIID^Gerät 1 (EtherCAT)^Klemme 1 (EK1200)^Klemme 3 (EL3446)^I4 Channel^Current'}
	MDP5001_342_I4_Channel_Current_1							AT%I*  : REAL;
	{attribute 'TcLinkTo' := 'TIID^Gerät 1 (EtherCAT)^Klemme 1 (EK1200)^Klemme 3 (EL3446)^I4 Channel^Active Power'}
	MDP5001_342_I4_Channel_Active_Power_1						AT%I*  : REAL;
	{attribute 'TcLinkTo' := 'TIID^Gerät 1 (EtherCAT)^Klemme 1 (EK1200)^Klemme 3 (EL3446)^I4 Channel^Apparent Power'}
	MDP5001_342_I4_Channel_Apparent_Power_1					AT%I*  : REAL;
	{attribute 'TcLinkTo' := 'TIID^Gerät 1 (EtherCAT)^Klemme 1 (EK1200)^Klemme 3 (EL3446)^I4 Channel^Reactive Power Fundamental'}
	MDP5001_342_I4_Channel_Reactive_Power_Fundamental_1		AT%I*  : REAL;
	{attribute 'TcLinkTo' := 'TIID^Gerät 1 (EtherCAT)^Klemme 1 (EK1200)^Klemme 3 (EL3446)^I4 Channel^Active Energy'}
	MDP5001_342_I4_Channel_Active_Energy_1					AT%I*  : DINT;
	{attribute 'TcLinkTo' := 'TIID^Gerät 1 (EtherCAT)^Klemme 1 (EK1200)^Klemme 3 (EL3446)^I5 Channel^Overcurrent'}
	MDP5001_342_I5_Channel_Overcurrent_1						AT%I*  : BOOL;
	{attribute 'TcLinkTo' := 'TIID^Gerät 1 (EtherCAT)^Klemme 1 (EK1200)^Klemme 3 (EL3446)^I5 Channel^Inaccurate Current'}
	MDP5001_342_I5_Channel_Inaccurate_Current_1				AT%I*  : BOOL;
	{attribute 'TcLinkTo' := 'TIID^Gerät 1 (EtherCAT)^Klemme 1 (EK1200)^Klemme 3 (EL3446)^I5 Channel^Current Guard Warning'}
	MDP5001_342_I5_Channel_Current_Guard_Warning_1			AT%I*  : bool;
	{attribute 'TcLinkTo' := 'TIID^Gerät 1 (EtherCAT)^Klemme 1 (EK1200)^Klemme 3 (EL3446)^I5 Channel^Current Guard Error'}
	MDP5001_342_I5_Channel_Current_Guard_Error_1				AT%I*  : bool;
	{attribute 'TcLinkTo' := 'TIID^Gerät 1 (EtherCAT)^Klemme 1 (EK1200)^Klemme 3 (EL3446)^I5 Channel^Apparent Power Guard Warning'}
	MDP5001_342_I5_Channel_Apparent_Power_Guard_Warning_1		AT%I*  : bool;
	{attribute 'TcLinkTo' := 'TIID^Gerät 1 (EtherCAT)^Klemme 1 (EK1200)^Klemme 3 (EL3446)^I5 Channel^Apparent Power Guard Error'}
	MDP5001_342_I5_Channel_Apparent_Power_Guard_Error_1		AT%I*  : bool;
	{attribute 'TcLinkTo' := 'TIID^Gerät 1 (EtherCAT)^Klemme 1 (EK1200)^Klemme 3 (EL3446)^I5 Channel^Active Power Guard Warning'}
	MDP5001_342_I5_Channel_Active_Power_Guard_Warning_1		AT%I*  : bool;
	{attribute 'TcLinkTo' := 'TIID^Gerät 1 (EtherCAT)^Klemme 1 (EK1200)^Klemme 3 (EL3446)^I5 Channel^Active Power Guard Error'}
	MDP5001_342_I5_Channel_Active_Power_Guard_Error_1			AT%I*  : bool;
	{attribute 'TcLinkTo' := 'TIID^Gerät 1 (EtherCAT)^Klemme 1 (EK1200)^Klemme 3 (EL3446)^I5 Channel^Reactive Power Guard Warning'}
	MDP5001_342_I5_Channel_Reactive_Power_Guard_Warning_1		AT%I*  : bool;
	{attribute 'TcLinkTo' := 'TIID^Gerät 1 (EtherCAT)^Klemme 1 (EK1200)^Klemme 3 (EL3446)^I5 Channel^Reactive Power Guard Error'}
	MDP5001_342_I5_Channel_Reactive_Power_Guard_Error_1		AT%I*  : bool;
	{attribute 'TcLinkTo' := 'TIID^Gerät 1 (EtherCAT)^Klemme 1 (EK1200)^Klemme 3 (EL3446)^I5 Channel^DPM Inaccurate'}
	MDP5001_342_I5_Channel_DPM_Inaccurate_1					AT%I*  : bool;
	{attribute 'TcLinkTo' := 'TIID^Gerät 1 (EtherCAT)^Klemme 1 (EK1200)^Klemme 3 (EL3446)^I5 Channel^DPM Timeout'}
	MDP5001_342_I5_Channel_DPM_Timeout_1						AT%I*  : bool;
	{attribute 'TcLinkTo' := 'TIID^Gerät 1 (EtherCAT)^Klemme 1 (EK1200)^Klemme 3 (EL3446)^I5 Channel^TxPDO Toggle'}
	MDP5001_342_I5_Channel_TxPDO_Toggle_1						AT%I*  : bool;
	{attribute 'TcLinkTo' := 'TIID^Gerät 1 (EtherCAT)^Klemme 1 (EK1200)^Klemme 3 (EL3446)^I5 Channel^Current'}
	MDP5001_342_I5_Channel_Current_1							AT%I*  : REAL;
	{attribute 'TcLinkTo' := 'TIID^Gerät 1 (EtherCAT)^Klemme 1 (EK1200)^Klemme 3 (EL3446)^I5 Channel^Active Power'}
	MDP5001_342_I5_Channel_Active_Power_1						AT%I*  : REAL;
	{attribute 'TcLinkTo' := 'TIID^Gerät 1 (EtherCAT)^Klemme 1 (EK1200)^Klemme 3 (EL3446)^I5 Channel^Apparent Power'}
	MDP5001_342_I5_Channel_Apparent_Power_1					AT%I*  : REAL;
	{attribute 'TcLinkTo' := 'TIID^Gerät 1 (EtherCAT)^Klemme 1 (EK1200)^Klemme 3 (EL3446)^I5 Channel^Reactive Power Fundamental'}
	MDP5001_342_I5_Channel_Reactive_Power_Fundamental_1		AT%I*  : REAL;
	{attribute 'TcLinkTo' := 'TIID^Gerät 1 (EtherCAT)^Klemme 1 (EK1200)^Klemme 3 (EL3446)^I5 Channel^Active Energy'}
	MDP5001_342_I5_Channel_Active_Energy_1					AT%I*  : DINT;
	{attribute 'TcLinkTo' := 'TIID^Gerät 1 (EtherCAT)^Klemme 1 (EK1200)^Klemme 3 (EL3446)^I6 Channel^Overcurrent'}
	MDP5001_342_I6_Channel_Overcurrent_1						AT%I*  : BOOL;
	{attribute 'TcLinkTo' := 'TIID^Gerät 1 (EtherCAT)^Klemme 1 (EK1200)^Klemme 3 (EL3446)^I6 Channel^Inaccurate Current'}
	MDP5001_342_I6_Channel_Inaccurate_Current_1				AT%I*  : BOOL;
	{attribute 'TcLinkTo' := 'TIID^Gerät 1 (EtherCAT)^Klemme 1 (EK1200)^Klemme 3 (EL3446)^I6 Channel^Current Guard Warning'}
	MDP5001_342_I6_Channel_Current_Guard_Warning_1			AT%I*  : bool;
	{attribute 'TcLinkTo' := 'TIID^Gerät 1 (EtherCAT)^Klemme 1 (EK1200)^Klemme 3 (EL3446)^I6 Channel^Current Guard Error'}
	MDP5001_342_I6_Channel_Current_Guard_Error_1				AT%I*  : bool;
	{attribute 'TcLinkTo' := 'TIID^Gerät 1 (EtherCAT)^Klemme 1 (EK1200)^Klemme 3 (EL3446)^I6 Channel^Apparent Power Guard Warning'}
	MDP5001_342_I6_Channel_Apparent_Power_Guard_Warning_1		AT%I*  : bool;
	{attribute 'TcLinkTo' := 'TIID^Gerät 1 (EtherCAT)^Klemme 1 (EK1200)^Klemme 3 (EL3446)^I6 Channel^Apparent Power Guard Error'}
	MDP5001_342_I6_Channel_Apparent_Power_Guard_Error_1		AT%I*  : bool;
	{attribute 'TcLinkTo' := 'TIID^Gerät 1 (EtherCAT)^Klemme 1 (EK1200)^Klemme 3 (EL3446)^I6 Channel^Active Power Guard Warning'}
	MDP5001_342_I6_Channel_Active_Power_Guard_Warning_1		AT%I*  : bool;
	{attribute 'TcLinkTo' := 'TIID^Gerät 1 (EtherCAT)^Klemme 1 (EK1200)^Klemme 3 (EL3446)^I6 Channel^Active Power Guard Error'}
	MDP5001_342_I6_Channel_Active_Power_Guard_Error_1			AT%I*  : bool;
	{attribute 'TcLinkTo' := 'TIID^Gerät 1 (EtherCAT)^Klemme 1 (EK1200)^Klemme 3 (EL3446)^I6 Channel^Reactive Power Guard Warning'}
	MDP5001_342_I6_Channel_Reactive_Power_Guard_Warning_1		AT%I*  : bool;
	{attribute 'TcLinkTo' := 'TIID^Gerät 1 (EtherCAT)^Klemme 1 (EK1200)^Klemme 3 (EL3446)^I6 Channel^Reactive Power Guard Error'}
	MDP5001_342_I6_Channel_Reactive_Power_Guard_Error_1		AT%I*  : bool;
	{attribute 'TcLinkTo' := 'TIID^Gerät 1 (EtherCAT)^Klemme 1 (EK1200)^Klemme 3 (EL3446)^I6 Channel^DPM Inaccurate'}
	MDP5001_342_I6_Channel_DPM_Inaccurate_1					AT%I*  : bool;
	{attribute 'TcLinkTo' := 'TIID^Gerät 1 (EtherCAT)^Klemme 1 (EK1200)^Klemme 3 (EL3446)^I6 Channel^DPM Timeout'}
	MDP5001_342_I6_Channel_DPM_Timeout_1						AT%I*  : bool;
	{attribute 'TcLinkTo' := 'TIID^Gerät 1 (EtherCAT)^Klemme 1 (EK1200)^Klemme 3 (EL3446)^I6 Channel^TxPDO Toggle'}
	MDP5001_342_I6_Channel_TxPDO_Toggle_1						AT%I*  : bool;
	{attribute 'TcLinkTo' := 'TIID^Gerät 1 (EtherCAT)^Klemme 1 (EK1200)^Klemme 3 (EL3446)^I6 Channel^Current'}
	MDP5001_342_I6_Channel_Current_1							AT%I*  : REAL;
	{attribute 'TcLinkTo' := 'TIID^Gerät 1 (EtherCAT)^Klemme 1 (EK1200)^Klemme 3 (EL3446)^I6 Channel^Active Power'}
	MDP5001_342_I6_Channel_Active_Power_1						AT%I*  : REAL;
	{attribute 'TcLinkTo' := 'TIID^Gerät 1 (EtherCAT)^Klemme 1 (EK1200)^Klemme 3 (EL3446)^I6 Channel^Apparent Power'}
	MDP5001_342_I6_Channel_Apparent_Power_1					AT%I*  : REAL;
	{attribute 'TcLinkTo' := 'TIID^Gerät 1 (EtherCAT)^Klemme 1 (EK1200)^Klemme 3 (EL3446)^I6 Channel^Reactive Power Fundamental'}
	MDP5001_342_I6_Channel_Reactive_Power_Fundamental_1		AT%I*  : REAL;
	{attribute 'TcLinkTo' := 'TIID^Gerät 1 (EtherCAT)^Klemme 1 (EK1200)^Klemme 3 (EL3446)^I6 Channel^Active Energy'}
	MDP5001_342_I6_Channel_Active_Energy_1					AT%I*  : DINT;	
	
	{attribute 'TcLinkTo' := 'TIID^Gerät 1 (EtherCAT)^Klemme 1 (EK1200)^Klemme 3 (EL3446)^DPM Variant Value In^TxPDO Toggle'}
	MDP5001_342_DPM_Variant_Value_In_TxPDO_Toggle_1			AT%I*  : BOOL;
	{attribute 'TcLinkTo' := 'TIID^Gerät 1 (EtherCAT)^Klemme 1 (EK1200)^Klemme 3 (EL3446)^DPM Variant Value In^Index 1 REAL'}
	MDP5001_342_DPM_Variant_Value_In_Index_1_REAL_1			AT%I*  : UINT;
	{attribute 'TcLinkTo' := 'TIID^Gerät 1 (EtherCAT)^Klemme 1 (EK1200)^Klemme 3 (EL3446)^DPM Variant Value In^Value 1 REAL'}
	MDP5001_342_DPM_Variant_Value_In_Value_1_REAL_1			AT%I*  : REAL;
	{attribute 'TcLinkTo' := 'TIID^Gerät 1 (EtherCAT)^Klemme 1 (EK1200)^Klemme 3 (EL3446)^DPM Variant Value In^Index 2 REAL'}
	MDP5001_342_DPM_Variant_Value_In_Index_2_REAL_1			AT%I*  : UINT;
	{attribute 'TcLinkTo' := 'TIID^Gerät 1 (EtherCAT)^Klemme 1 (EK1200)^Klemme 3 (EL3446)^DPM Variant Value In^Value 2 REAL'}
	MDP5001_342_DPM_Variant_Value_In_Value_2_REAL_1			AT%I*  : REAL;
	{attribute 'TcLinkTo' := 'TIID^Gerät 1 (EtherCAT)^Klemme 1 (EK1200)^Klemme 3 (EL3446)^DPM Variant Value In^Index 3 REAL'}
	MDP5001_342_DPM_Variant_Value_In_Index_3_REAL_1			AT%I*  : UINT;
	{attribute 'TcLinkTo' := 'TIID^Gerät 1 (EtherCAT)^Klemme 1 (EK1200)^Klemme 3 (EL3446)^DPM Variant Value In^Value 3 REAL'}
	MDP5001_342_DPM_Variant_Value_In_Value_3_REAL_1			AT%I*  : REAL;
	{attribute 'TcLinkTo' := 'TIID^Gerät 1 (EtherCAT)^Klemme 1 (EK1200)^Klemme 3 (EL3446)^DPM Variant Value In^Index 4 ULINT'}
	MDP5001_342_DPM_Variant_Value_In_Index_4_ULINT_1			AT%I*  : UINT;
	{attribute 'TcLinkTo' := 'TIID^Gerät 1 (EtherCAT)^Klemme 1 (EK1200)^Klemme 3 (EL3446)^DPM Variant Value In^Value 4 ULINT'}
	MDP5001_342_DPM_Variant_Value_In_Value_4_ULINT_1			AT%I*  : ULINT;

	{attribute 'TcLinkTo' := 'TIID^Gerät 1 (EtherCAT)^Klemme 1 (EK1200)^Klemme 3 (EL3446)^DPM Variant Value Out^Index 1 REAL'}
	MDP5001_342_DPM_Variant_Value_Out_Index_1_REAL_1	AT%Q* : UINT;
	{attribute 'TcLinkTo' := 'TIID^Gerät 1 (EtherCAT)^Klemme 1 (EK1200)^Klemme 3 (EL3446)^DPM Variant Value Out^Index 2 REAL'}
	MDP5001_342_DPM_Variant_Value_Out_Index_2_REAL_1	AT%Q* : UINT;
	{attribute 'TcLinkTo' := 'TIID^Gerät 1 (EtherCAT)^Klemme 1 (EK1200)^Klemme 3 (EL3446)^DPM Variant Value Out^Index 3 REAL'}
	MDP5001_342_DPM_Variant_Value_Out_Index_3_REAL_1	AT%Q* : UINT;
	{attribute 'TcLinkTo' := 'TIID^Gerät 1 (EtherCAT)^Klemme 1 (EK1200)^Klemme 3 (EL3446)^DPM Variant Value Out^Index 4 ULINT'}
	MDP5001_342_DPM_Variant_Value_Out_Index_4_ULINT_1	AT%Q* : UINT;
	{attribute 'TcLinkTo' := 'TIID^Gerät 1 (EtherCAT)^Klemme 1 (EK1200)^Klemme 3 (EL3446)^DPM Data^Data 1'}
	MDP5001_342_DPM_Data_Data_1_1						AT%Q* : UDINT;
	{attribute 'TcLinkTo' := 'TIID^Gerät 1 (EtherCAT)^Klemme 1 (EK1200)^Klemme 3 (EL3446)^DPM Data^Data 2'}
	MDP5001_342_DPM_Data_Data_2_1						AT%Q* : UDINT;
	{attribute 'TcLinkTo' := 'TIID^Gerät 1 (EtherCAT)^Klemme 1 (EK1200)^Klemme 3 (EL3446)^DPM Data^Data 3'}
	MDP5001_342_DPM_Data_Data_3_1						AT%Q* : UDINT;
	{attribute 'TcLinkTo' := 'TIID^Gerät 1 (EtherCAT)^Klemme 1 (EK1200)^Klemme 3 (EL3446)^DPM Data^Data 4'}
	MDP5001_342_DPM_Data_Data_4_1						AT%Q* : UDINT;
	{attribute 'TcLinkTo' := 'TIID^Gerät 1 (EtherCAT)^Klemme 1 (EK1200)^Klemme 3 (EL3446)^DPM Data^Data 5'}
	MDP5001_342_DPM_Data_Data_5_1						AT%Q* : UDINT;
	{attribute 'TcLinkTo' := 'TIID^Gerät 1 (EtherCAT)^Klemme 1 (EK1200)^Klemme 3 (EL3446)^DPM Data^Data 6'}
	MDP5001_342_DPM_Data_Data_6_1						AT%Q* : UDINT;
	{attribute 'TcLinkTo' := 'TIID^Gerät 1 (EtherCAT)^Klemme 1 (EK1200)^Klemme 3 (EL3446)^DPM Data^Data 7'}
	MDP5001_342_DPM_Data_Data_7_1						AT%Q* : UDINT;
	{attribute 'TcLinkTo' := 'TIID^Gerät 1 (EtherCAT)^Klemme 1 (EK1200)^Klemme 3 (EL3446)^DPM Data^Data 8'}
	MDP5001_342_DPM_Data_Data_8_1						AT%Q* : UDINT;
	{attribute 'TcLinkTo' := 'TIID^Gerät 1 (EtherCAT)^Klemme 1 (EK1200)^Klemme 3 (EL3446)^DPM Data^Data 9'}
	MDP5001_342_DPM_Data_Data_9_1						AT%Q* : UDINT;
	{attribute 'TcLinkTo' := 'TIID^Gerät 1 (EtherCAT)^Klemme 1 (EK1200)^Klemme 3 (EL3446)^DPM Data^Data 10'}
	MDP5001_342_DPM_Data_Data_10_1					AT%Q* : UDINT;
	{attribute 'TcLinkTo' := 'TIID^Gerät 1 (EtherCAT)^Klemme 1 (EK1200)^Klemme 3 (EL3446)^DPM Data^Data 11'}
	MDP5001_342_DPM_Data_Data_11_1					AT%Q* : UDINT;
	{attribute 'TcLinkTo' := 'TIID^Gerät 1 (EtherCAT)^Klemme 1 (EK1200)^Klemme 3 (EL3446)^DPM Data^Data 12'}
	MDP5001_342_DPM_Data_Data_12_1					AT%Q* : UDINT;
	{attribute 'TcLinkTo' := 'TIID^Gerät 1 (EtherCAT)^Klemme 1 (EK1200)^Klemme 3 (EL3446)^DPM Data^Data 13'}
	MDP5001_342_DPM_Data_Data_13_1					AT%Q* : UDINT;
	{attribute 'TcLinkTo' := 'TIID^Gerät 1 (EtherCAT)^Klemme 1 (EK1200)^Klemme 3 (EL3446)^DPM Data^Data 14'}
	MDP5001_342_DPM_Data_Data_14_1					AT%Q* : UDINT;
	{attribute 'TcLinkTo' := 'TIID^Gerät 1 (EtherCAT)^Klemme 1 (EK1200)^Klemme 3 (EL3446)^DPM Data^Data 15'}
	MDP5001_342_DPM_Data_Data_15_1					AT%Q* : UDINT;
	{attribute 'TcLinkTo' := 'TIID^Gerät 1 (EtherCAT)^Klemme 1 (EK1200)^Klemme 3 (EL3446)^DPM Data^Data 16'}
	MDP5001_342_DPM_Data_Data_16_1					AT%Q* : UDINT;
	{attribute 'TcLinkTo' := 'TIID^Gerät 1 (EtherCAT)^Klemme 1 (EK1200)^Klemme 3 (EL3446)^DPM Data^Data 17'}
	MDP5001_342_DPM_Data_Data_17_1					AT%Q* : UDINT;
	{attribute 'TcLinkTo' := 'TIID^Gerät 1 (EtherCAT)^Klemme 1 (EK1200)^Klemme 3 (EL3446)^DPM Data^Data 18'}
	MDP5001_342_DPM_Data_Data_18_1					AT%Q* : UDINT;
	{attribute 'TcLinkTo' := 'TIID^Gerät 1 (EtherCAT)^Klemme 1 (EK1200)^Klemme 3 (EL3446)^DPM Data^Data 19'}
	MDP5001_342_DPM_Data_Data_19_1					AT%Q* : UDINT;
	{attribute 'TcLinkTo' := 'TIID^Gerät 1 (EtherCAT)^Klemme 1 (EK1200)^Klemme 3 (EL3446)^DPM Data^Data 20'}
	MDP5001_342_DPM_Data_Data_20_1					AT%Q* : UDINT;



